LIN {X 0,Y 193.784,Z 1192.753,A -85,B 0,C 180,E1 2958.088,E2 2958.088} C_VEL
LIN {X 0,Y 196.55,Z 1189.097,A -85,B 0,C 180,E1 2951.921,E2 2951.921} C_VEL
LIN {X 0,Y 200.863,Z 1184.423,A -85,B 0,C 180,E1 2945.908,E2 2945.908} C_VEL
LIN {X 0,Y 207.135,Z 1178.405,A -85,B 0,C 180,E1 2939.865,E2 2939.865} C_VEL
LIN {X 0,Y 216.126,Z 1170.427,A -85,B 0,C 180,E1 2933.611,E2 2933.611} C_VEL
LIN {X 0,Y 228.412,Z 1159.714,A -85,B 0,C 180,E1 2927.271,E2 2927.271} C_VEL
LIN {X 0,Y 240.181,Z 1149.383,A -85,B 0,C 180,E1 2922.535,E2 2922.535} C_VEL
LIN {X 0,Y 252.062,Z 1138.725,A -85,B 0,C 180,E1 2918.605,E2 2918.605} C_VEL
LIN {X 0,Y 266.276,Z 1125.508,A -85,B 0,C 180,E1 2914.678,E2 2914.678} C_VEL
LIN {X 0,Y 283.027,Z 1108.844,A -85,B 0,C 180,E1 2910.815,E2 2910.815} C_VEL
LIN {X 0,Y 296.928,Z 1094.045,A -85,B 0,C 180,E1 2908.083,E2 2908.083} C_VEL
LIN {X 0,Y 310.128,Z 1079.059,A -85,B 0,C 180,E1 2905.802,E2 2905.802} C_VEL
LIN {X 0,Y 325.384,Z 1060.451,A -85,B 0,C 180,E1 2903.47,E2 2903.47} C_VEL
LIN {X 0,Y 340.885,Z 1039.444,A -85,B 0,C 180,E1 2901.363,E2 2901.363} C_VEL
LIN {X 0,Y 353.003,Z 1021.479,A -85,B 0,C 180,E1 2899.882,E2 2899.882} C_VEL
LIN {X 0,Y 363.602,Z 1004.327,A -85,B 0,C 180,E1 2898.674,E2 2898.674} C_VEL
LIN {X 0,Y 374.359,Z 985.261,A -85,B 0,C 180,E1 2897.538,E2 2897.538} C_VEL
LIN {X 0,Y 386.572,Z 961.109,A -85,B 0,C 180,E1 2896.341,E2 2896.341} C_VEL
LIN {X 0,Y 397.152,Z 936.648,A -85,B 0,C 180,E1 2895.366,E2 2895.366} C_VEL
LIN {X 0,Y 404.715,Z 916.743,A -85,B 0,C 180,E1 2894.708,E2 2894.708} C_VEL
LIN {X 0,Y 411.43,Z 896.473,A -85,B 0,C 180,E1 2894.146,E2 2894.146} C_VEL
LIN {X 0,Y 417.527,Z 874.884,A -85,B 0,C 180,E1 2893.651,E2 2893.651} C_VEL
LIN {X 0,Y 423.796,Z 847.505,A -85,B 0,C 180,E1 2893.158,E2 2893.158} C_VEL
LIN {X 0,Y 428.05,Z 821.26,A -85,B 0,C 180,E1 2892.768,E2 2892.768} C_VEL
LIN {X 0,Y 447.316,Z 647.119,A -85,B 0,C 180,E1 2890.414,E2 2890.414} C_VEL
LIN {X 0,Y 447.378,Z 646.28,A -85,B 0,C 180,E1 2890.372,E2 2890.372} C_VEL
LIN {X 0,Y 445.988,Z 643.083,A -85,B 0,C 180,E1 2888.25,E2 2888.25} C_VEL
LIN {X 0,Y 444.811,Z 639.498,A -85,B 0,C 180,E1 2884.758,E2 2884.758} C_VEL
LIN {X 0,Y 444.548,Z 640.357,A -85,B 0,C 180,E1 2883.764,E2 2883.764} C_VEL
LIN {X 0,Y 444.064,Z 644.495,A -85,B 0,C 180,E1 2882.115,E2 2882.115} C_VEL
LIN {X 0,Y 443.95,Z 648.203,A -85,B 0,C 180,E1 2880.587,E2 2880.587} C_VEL
LIN {X 0,Y 444,Z 648.603,A -85,B 0,C 180,E1 2880.301,E2 2880.301} C_VEL
LIN {X 0,Y 445.315,Z 651.864,A -85,B 0,C 180,E1 2877.297,E2 2877.297} C_VEL
LIN {X 0,Y 445.715,Z 653.234,A -85,B 0,C 180,E1 2876.601,E2 2876.601} C_VEL
LIN {X 0,Y 426.682,Z 822.591,A -85,B 0,C 180,E1 2874.347,E2 2874.347} C_VEL
LIN {X 0,Y 422.446,Z 848.515,A -85,B 0,C 180,E1 2873.967,E2 2873.967} C_VEL
LIN {X 0,Y 416.03,Z 876.307,A -85,B 0,C 180,E1 2873.503,E2 2873.503} C_VEL
LIN {X 0,Y 409.724,Z 898.303,A -85,B 0,C 180,E1 2873.036,E2 2873.036} C_VEL
LIN {X 0,Y 402.64,Z 919.334,A -85,B 0,C 180,E1 2872.488,E2 2872.488} C_VEL
LIN {X 0,Y 393.996,Z 941.562,A -85,B 0,C 180,E1 2871.786,E2 2871.786} C_VEL
LIN {X 0,Y 381.931,Z 968.144,A -85,B 0,C 180,E1 2870.742,E2 2870.742} C_VEL
LIN {X 0,Y 371.433,Z 988.383,A -85,B 0,C 180,E1 2869.766,E2 2869.766} C_VEL
LIN {X 0,Y 360.939,Z 1006.691,A -85,B 0,C 180,E1 2868.714,E2 2868.714} C_VEL
LIN {X 0,Y 349.835,Z 1024.338,A -85,B 0,C 180,E1 2867.527,E2 2867.527} C_VEL
LIN {X 0,Y 336.067,Z 1044.358,A -85,B 0,C 180,E1 2865.914,E2 2865.914} C_VEL
LIN {X 0,Y 319.422,Z 1066.078,A -85,B 0,C 180,E1 2863.734,E2 2863.734} C_VEL
LIN {X 0,Y 305.681,Z 1082.487,A -85,B 0,C 180,E1 2861.698,E2 2861.698} C_VEL
LIN {X 0,Y 292.491,Z 1097.171,A -85,B 0,C 180,E1 2859.501,E2 2859.501} C_VEL
LIN {X 0,Y 278.409,Z 1111.856,A -85,B 0,C 180,E1 2856.839,E2 2856.839} C_VEL
LIN {X 0,Y 260.253,Z 1129.443,A -85,B 0,C 180,E1 2852.794,E2 2852.794} C_VEL
LIN {X 0,Y 246.812,Z 1141.663,A -85,B 0,C 180,E1 2849.189,E2 2849.189} C_VEL
LIN {X 0,Y 234.676,Z 1152.282,A -85,B 0,C 180,E1 2845.318,E2 2845.318} C_VEL
LIN {X 0,Y 222.868,Z 1162.354,A -85,B 0,C 180,E1 2840.758,E2 2840.758} C_VEL
LIN {X 0,Y 210.031,Z 1173.278,A -85,B 0,C 180,E1 2834.413,E2 2834.413} C_VEL
LIN {X 0,Y 199.904,Z 1181.947,A -85,B 0,C 180,E1 2827.607,E2 2827.607} C_VEL
LIN {X 0,Y 193.365,Z 1187.998,A -85,B 0,C 180,E1 2821.485,E2 2821.485} C_VEL
LIN {X 0,Y 188.86,Z 1192.711,A -85,B 0,C 180,E1 2815.395,E2 2815.395} C_VEL
LIN {X 0,Y 185.836,Z 1196.591,A -85,B 0,C 180,E1 2808.835,E2 2808.835} C_VEL
LIN {X 0,Y 184.378,Z 1199.289,A -85,B 0,C 180,E1 2802.529,E2 2802.529} C_VEL
LIN {X 0,Y 183.967,Z 1200.898,A -85,B 0,C 180,E1 2796.869,E2 2796.869} C_VEL
LIN {X 0,Y 183.92,Z 1201.731,A -85,B 0,C 180,E1 2791.559,E2 2791.559} C_VEL
LIN {X 0,Y 183.915,Z 1201.914,A -85,B 0,C 180,E1 2786.261,E2 2786.261} C_VEL
LIN {X 0,Y 184.128,Z 1201.247,A -85,B 0,C 180,E1 2779.994,E2 2779.994} C_VEL
LIN {X 0,Y 185.319,Z 1199.444,A -85,B 0,C 180,E1 2773.062,E2 2773.062} C_VEL
LIN {X 0,Y 188.166,Z 1196.498,A -85,B 0,C 180,E1 2766.063,E2 2766.063} C_VEL
LIN {X 0,Y 192.831,Z 1192.57,A -85,B 0,C 180,E1 2759.46,E2 2759.46} C_VEL
LIN {X 0,Y 199.23,Z 1187.715,A -85,B 0,C 180,E1 2753.33,E2 2753.33} C_VEL
LIN {X 0,Y 208.339,Z 1181.197,A -85,B 0,C 180,E1 2747.041,E2 2747.041} C_VEL
LIN {X 0,Y 222.726,Z 1171.072,A -85,B 0,C 180,E1 2739.857,E2 2739.857} C_VEL
LIN {X 0,Y 236.169,Z 1161.389,A -85,B 0,C 180,E1 2734.782,E2 2734.782} C_VEL
LIN {X 0,Y 249.143,Z 1151.762,A -85,B 0,C 180,E1 2730.816,E2 2730.816} C_VEL
LIN {X 0,Y 263.881,Z 1140.338,A -85,B 0,C 180,E1 2727.073,E2 2727.073} C_VEL
LIN {X 0,Y 282.835,Z 1124.684,A -85,B 0,C 180,E1 2723.105,E2 2723.105} C_VEL
LIN {X 0,Y 299.39,Z 1109.822,A -85,B 0,C 180,E1 2720.208,E2 2720.208} C_VEL
LIN {X 0,Y 314.262,Z 1095.515,A -85,B 0,C 180,E1 2717.954,E2 2717.954} C_VEL
LIN {X 0,Y 329.586,Z 1079.656,A -85,B 0,C 180,E1 2715.913,E2 2715.913} C_VEL
LIN {X 0,Y 347.949,Z 1058.826,A -85,B 0,C 180,E1 2713.767,E2 2713.767} C_VEL
LIN {X 0,Y 362.448,Z 1040.568,A -85,B 0,C 180,E1 2712.264,E2 2712.264} C_VEL
LIN {X 0,Y 375.061,Z 1023.222,A -85,B 0,C 180,E1 2711.067,E2 2711.067} C_VEL
LIN {X 0,Y 387.331,Z 1004.748,A -85,B 0,C 180,E1 2710,E2 2710} C_VEL
LIN {X 0,Y 399.863,Z 983.893,A -85,B 0,C 180,E1 2708.994,E2 2708.994} C_VEL
LIN {X 0,Y 413.455,Z 958.023,A -85,B 0,C 180,E1 2707.988,E2 2707.988} C_VEL
LIN {X 0,Y 422.9,Z 937.408,A -85,B 0,C 180,E1 2707.335,E2 2707.335} C_VEL
LIN {X 0,Y 431.26,Z 916.643,A -85,B 0,C 180,E1 2706.791,E2 2706.791} C_VEL
LIN {X 0,Y 438.618,Z 895.545,A -85,B 0,C 180,E1 2706.334,E2 2706.334} C_VEL
LIN {X 0,Y 446.408,Z 868.875,A -85,B 0,C 180,E1 2705.874,E2 2705.874} C_VEL
LIN {X 0,Y 452.306,Z 842.166,A -85,B 0,C 180,E1 2705.505,E2 2705.505} C_VEL
LIN {X 0,Y 456.042,Z 819.713,A -85,B 0,C 180,E1 2705.211,E2 2705.211} C_VEL
LIN {X 0,Y 473.449,Z 676.945,A -85,B 0,C 180,E1 2703.423,E2 2703.423} C_VEL
LIN {X 0,Y 473.466,Z 676.653,A -85,B 0,C 180,E1 2702.713,E2 2702.713} C_VEL
LIN {X 0,Y 473.43,Z 677.084,A -85,B 0,C 180,E1 2702.407,E2 2702.407} C_VEL
LIN {X 0,Y 455.697,Z 821.974,A -85,B 0,C 180,E1 2700.598,E2 2700.598} C_VEL
LIN {X 0,Y 450.971,Z 849.012,A -85,B 0,C 180,E1 2700.243,E2 2700.243} C_VEL
LIN {X 0,Y 444.348,Z 875.944,A -85,B 0,C 180,E1 2699.835,E2 2699.835} C_VEL
LIN {X 0,Y 437.962,Z 897.143,A -85,B 0,C 180,E1 2699.43,E2 2699.43} C_VEL
LIN {X 0,Y 430.703,Z 917.681,A -85,B 0,C 180,E1 2698.954,E2 2698.954} C_VEL
LIN {X 0,Y 422.114,Z 938.76,A -85,B 0,C 180,E1 2698.367,E2 2698.367} C_VEL
LIN {X 0,Y 409.93,Z 964.599,A -85,B 0,C 180,E1 2697.484,E2 2697.484} C_VEL
LIN {X 0,Y 398.155,Z 986.144,A -85,B 0,C 180,E1 2696.577,E2 2696.577} C_VEL
LIN {X 0,Y 387.061,Z 1004.427,A -85,B 0,C 180,E1 2695.652,E2 2695.652} C_VEL
LIN {X 0,Y 375.114,Z 1022.302,A -85,B 0,C 180,E1 2694.599,E2 2694.599} C_VEL
LIN {X 0,Y 361.439,Z 1040.964,A -85,B 0,C 180,E1 2693.273,E2 2693.273} C_VEL
LIN {X 0,Y 343.377,Z 1063.103,A -85,B 0,C 180,E1 2691.329,E2 2691.329} C_VEL
LIN {X 0,Y 328.434,Z 1079.641,A -85,B 0,C 180,E1 2689.52,E2 2689.52} C_VEL
LIN {X 0,Y 314.281,Z 1094.13,A -85,B 0,C 180,E1 2687.606,E2 2687.606} C_VEL
LIN {X 0,Y 299.083,Z 1108.599,A -85,B 0,C 180,E1 2685.281,E2 2685.281} C_VEL
LIN {X 0,Y 280.33,Z 1125.143,A -85,B 0,C 180,E1 2681.922,E2 2681.922} C_VEL
LIN {X 0,Y 263.578,Z 1138.659,A -85,B 0,C 180,E1 2678.339,E2 2678.339} C_VEL
LIN {X 0,Y 249.729,Z 1149.238,A -85,B 0,C 180,E1 2674.803,E2 2674.803} C_VEL
LIN {X 0,Y 236.884,Z 1158.604,A -85,B 0,C 180,E1 2670.894,E2 2670.894} C_VEL
LIN {X 0,Y 223.454,Z 1168.069,A -85,B 0,C 180,E1 2665.872,E2 2665.872} C_VEL
LIN {X 0,Y 209.417,Z 1177.701,A -85,B 0,C 180,E1 2658.969,E2 2658.969} C_VEL
LIN {X 0,Y 200.157,Z 1184.082,A -85,B 0,C 180,E1 2652.748,E2 2652.748} C_VEL
LIN {X 0,Y 193.407,Z 1188.958,A -85,B 0,C 180,E1 2646.477,E2 2646.477} C_VEL
LIN {X 0,Y 188.589,Z 1192.766,A -85,B 0,C 180,E1 2639.891,E2 2639.891} C_VEL
LIN {X 0,Y 185.648,Z 1195.509,A -85,B 0,C 180,E1 2633.15,E2 2633.15} C_VEL
LIN {X 0,Y 184.261,Z 1197.282,A -85,B 0,C 180,E1 2626.065,E2 2626.065} C_VEL
LIN {X 0,Y 183.939,Z 1197.909,A -85,B 0,C 180,E1 2619.7,E2 2619.7} C_VEL
LIN {X 0,Y 183.918,Z 1197.682,A -85,B 0,C 180,E1 2614.052,E2 2614.052} C_VEL
LIN {X 0,Y 184.043,Z 1196.747,A -85,B 0,C 180,E1 2608.442,E2 2608.442} C_VEL
LIN {X 0,Y 184.659,Z 1194.997,A -85,B 0,C 180,E1 2602.532,E2 2602.532} C_VEL
LIN {X 0,Y 186.366,Z 1192.29,A -85,B 0,C 180,E1 2596.344,E2 2596.344} C_VEL
LIN {X 0,Y 189.631,Z 1188.474,A -85,B 0,C 180,E1 2589.956,E2 2589.956} C_VEL
LIN {X 0,Y 195.401,Z 1182.891,A -85,B 0,C 180,E1 2582.907,E2 2582.907} C_VEL
LIN {X 0,Y 204.952,Z 1174.56,A -85,B 0,C 180,E1 2575.193,E2 2575.193} C_VEL
LIN {X 0,Y 214.979,Z 1166.193,A -85,B 0,C 180,E1 2569.371,E2 2569.371} C_VEL
LIN {X 0,Y 225.673,Z 1157.324,A -85,B 0,C 180,E1 2564.492,E2 2564.492} C_VEL
LIN {X 0,Y 238.322,Z 1146.688,A -85,B 0,C 180,E1 2559.844,E2 2559.844} C_VEL
LIN {X 0,Y 254.991,Z 1132.046,A -85,B 0,C 180,E1 2554.925,E2 2554.925} C_VEL
LIN {X 0,Y 268.749,Z 1119.234,A -85,B 0,C 180,E1 2551.57,E2 2551.57} C_VEL
LIN {X 0,Y 281.856,Z 1106.336,A -85,B 0,C 180,E1 2548.808,E2 2548.808} C_VEL
LIN {X 0,Y 295.173,Z 1092.404,A -85,B 0,C 180,E1 2546.344,E2 2546.344} C_VEL
LIN {X 0,Y 311.307,Z 1074.339,A -85,B 0,C 180,E1 2543.739,E2 2543.739} C_VEL
LIN {X 0,Y 327.195,Z 1054.608,A -85,B 0,C 180,E1 2541.482,E2 2541.482} C_VEL
LIN {X 0,Y 340.141,Z 1037.088,A -85,B 0,C 180,E1 2539.834,E2 2539.834} C_VEL
LIN {X 0,Y 352.066,Z 1019.537,A -85,B 0,C 180,E1 2538.455,E2 2538.455} C_VEL
LIN {X 0,Y 364.175,Z 1000.011,A -85,B 0,C 180,E1 2537.162,E2 2537.162} C_VEL
LIN {X 0,Y 377.653,Z 975.504,A -85,B 0,C 180,E1 2535.826,E2 2535.826} C_VEL
LIN {X 0,Y 387.964,Z 954.171,A -85,B 0,C 180,E1 2534.879,E2 2534.879} C_VEL
LIN {X 0,Y 396.471,Z 934.374,A -85,B 0,C 180,E1 2534.143,E2 2534.143} C_VEL
LIN {X 0,Y 404.135,Z 914.142,A -85,B 0,C 180,E1 2533.509,E2 2533.509} C_VEL
LIN {X 0,Y 412.068,Z 889.833,A -85,B 0,C 180,E1 2532.879,E2 2532.879} C_VEL
LIN {X 0,Y 419.216,Z 862.435,A -85,B 0,C 180,E1 2532.33,E2 2532.33} C_VEL
LIN {X 0,Y 423.88,Z 839.666,A -85,B 0,C 180,E1 2531.97,E2 2531.97} C_VEL
LIN {X 0,Y 427.315,Z 817.269,A -85,B 0,C 180,E1 2531.649,E2 2531.649} C_VEL
LIN {X 0,Y 445.713,Z 652.932,A -85,B 0,C 180,E1 2529.458,E2 2529.458} C_VEL
LIN {X 0,Y 444.938,Z 650.967,A -85,B 0,C 180,E1 2528.139,E2 2528.139} C_VEL
LIN {X 0,Y 443.812,Z 647.425,A -85,B 0,C 180,E1 2524.652,E2 2524.652} C_VEL
LIN {X 0,Y 443.864,Z 647.551,A -85,B 0,C 180,E1 2521.162,E2 2521.162} C_VEL
LIN {X 0,Y 444,Z 648.603,A -85,B 0,C 180,E1 2520.301,E2 2520.301} C_VEL
LIN {X 0,Y 444.352,Z 650.816,A -85,B 0,C 180,E1 2518.94,E2 2518.94} C_VEL
LIN {X 0,Y 444.48,Z 653.384,A -85,B 0,C 180,E1 2518.202,E2 2518.202} C_VEL
LIN {X 0,Y 444.411,Z 656.348,A -85,B 0,C 180,E1 2517.767,E2 2517.767} C_VEL
LIN {X 0,Y 444.172,Z 659.579,A -85,B 0,C 180,E1 2517.547,E2 2517.547} C_VEL
LIN {X 0,Y 425.554,Z 822.606,A -85,B 0,C 180,E1 2515.415,E2 2515.415} C_VEL
LIN {X 0,Y 421.185,Z 848.96,A -85,B 0,C 180,E1 2515.039,E2 2515.039} C_VEL
LIN {X 0,Y 414.704,Z 876.574,A -85,B 0,C 180,E1 2514.592,E2 2514.592} C_VEL
LIN {X 0,Y 408.459,Z 898.118,A -85,B 0,C 180,E1 2514.152,E2 2514.152} C_VEL
LIN {X 0,Y 401.429,Z 918.8,A -85,B 0,C 180,E1 2513.634,E2 2513.634} C_VEL
LIN {X 0,Y 392.432,Z 941.7,A -85,B 0,C 180,E1 2512.937,E2 2512.937} C_VEL
LIN {X 0,Y 380.221,Z 968.234,A -85,B 0,C 180,E1 2511.93,E2 2511.93} C_VEL
LIN {X 0,Y 369.526,Z 988.564,A -85,B 0,C 180,E1 2510.981,E2 2510.981} C_VEL
LIN {X 0,Y 358.884,Z 1006.85,A -85,B 0,C 180,E1 2509.961,E2 2509.961} C_VEL
LIN {X 0,Y 347.571,Z 1024.544,A -85,B 0,C 180,E1 2508.808,E2 2508.808} C_VEL
LIN {X 0,Y 332.902,Z 1045.5,A -85,B 0,C 180,E1 2507.158,E2 2507.158} C_VEL
LIN {X 0,Y 316.333,Z 1066.583,A -85,B 0,C 180,E1 2505.075,E2 2505.075} C_VEL
LIN {X 0,Y 302.936,Z 1082.257,A -85,B 0,C 180,E1 2503.174,E2 2503.174} C_VEL
LIN {X 0,Y 289.651,Z 1096.737,A -85,B 0,C 180,E1 2501.06,E2 2501.06} C_VEL
LIN {X 0,Y 275.986,Z 1110.665,A -85,B 0,C 180,E1 2498.607,E2 2498.607} C_VEL
LIN {X 0,Y 259.115,Z 1126.81,A -85,B 0,C 180,E1 2495.071,E2 2495.071} C_VEL
LIN {X 0,Y 242.557,Z 1141.372,A -85,B 0,C 180,E1 2490.894,E2 2490.894} C_VEL
LIN {X 0,Y 229.971,Z 1151.986,A -85,B 0,C 180,E1 2487.05,E2 2487.05} C_VEL
LIN {X 0,Y 217.832,Z 1161.904,A -85,B 0,C 180,E1 2482.571,E2 2482.571} C_VEL
LIN {X 0,Y 204.987,Z 1172.328,A -85,B 0,C 180,E1 2476.546,E2 2476.546} C_VEL
LIN {X 0,Y 193.711,Z 1181.428,A -85,B 0,C 180,E1 2469.413,E2 2469.413} C_VEL
LIN {X 0,Y 186.602,Z 1187.549,A -85,B 0,C 180,E1 2463.132,E2 2463.132} C_VEL
LIN {X 0,Y 181.412,Z 1192.542,A -85,B 0,C 180,E1 2456.517,E2 2456.517} C_VEL
LIN {X 0,Y 178.201,Z 1196.278,A -85,B 0,C 180,E1 2450.016,E2 2450.016} C_VEL
LIN {X 0,Y 176.553,Z 1198.926,A -85,B 0,C 180,E1 2443.761,E2 2443.761} C_VEL
LIN {X 0,Y 176.006,Z 1200.647,A -85,B 0,C 180,E1 2437.837,E2 2437.837} C_VEL
LIN {X 0,Y 175.916,Z 1201.59,A -85,B 0,C 180,E1 2432.281,E2 2432.281} C_VEL
LIN {X 0,Y 175.915,Z 1201.858,A -85,B 0,C 180,E1 2426.417,E2 2426.417} C_VEL
LIN {X 0,Y 176.136,Z 1201.253,A -85,B 0,C 180,E1 2419.866,E2 2419.866} C_VEL
LIN {X 0,Y 177.562,Z 1199.335,A -85,B 0,C 180,E1 2412.116,E2 2412.116} C_VEL
LIN {X 0,Y 180.772,Z 1196.365,A -85,B 0,C 180,E1 2404.794,E2 2404.794} C_VEL
LIN {X 0,Y 185.712,Z 1192.557,A -85,B 0,C 180,E1 2398.156,E2 2398.156} C_VEL
LIN {X 0,Y 192.592,Z 1187.722,A -85,B 0,C 180,E1 2391.845,E2 2391.845} C_VEL
LIN {X 0,Y 201.817,Z 1181.526,A -85,B 0,C 180,E1 2385.69,E2 2385.69} C_VEL
LIN {X 0,Y 215.739,Z 1172.347,A -85,B 0,C 180,E1 2378.867,E2 2378.867} C_VEL
LIN {X 0,Y 230.84,Z 1161.935,A -85,B 0,C 180,E1 2373.285,E2 2373.285} C_VEL
LIN {X 0,Y 244.956,Z 1151.875,A -85,B 0,C 180,E1 2369.132,E2 2369.132} C_VEL
LIN {X 0,Y 259.673,Z 1140.865,A -85,B 0,C 180,E1 2365.548,E2 2365.548} C_VEL
LIN {X 0,Y 277.939,Z 1126.377,A -85,B 0,C 180,E1 2361.855,E2 2361.855} C_VEL
LIN {X 0,Y 296.631,Z 1110.043,A -85,B 0,C 180,E1 2358.707,E2 2358.707} C_VEL
LIN {X 0,Y 311.816,Z 1095.77,A -85,B 0,C 180,E1 2356.511,E2 2356.511} C_VEL
LIN {X 0,Y 326.549,Z 1080.856,A -85,B 0,C 180,E1 2354.634,E2 2354.634} C_VEL
LIN {X 0,Y 343.701,Z 1062.031,A -85,B 0,C 180,E1 2352.707,E2 2352.707} C_VEL
LIN {X 0,Y 360.601,Z 1041.239,A -85,B 0,C 180,E1 2351.021,E2 2351.021} C_VEL
LIN {X 0,Y 373.464,Z 1023.85,A -85,B 0,C 180,E1 2349.859,E2 2349.859} C_VEL
LIN {X 0,Y 386.012,Z 1005.253,A -85,B 0,C 180,E1 2348.82,E2 2348.82} C_VEL
LIN {X 0,Y 398.151,Z 985.373,A -85,B 0,C 180,E1 2347.892,E2 2347.892} C_VEL
LIN {X 0,Y 411.946,Z 959.743,A -85,B 0,C 180,E1 2346.921,E2 2346.921} C_VEL
LIN {X 0,Y 422.054,Z 938.014,A -85,B 0,C 180,E1 2346.256,E2 2346.256} C_VEL
LIN {X 0,Y 430.556,Z 917.171,A -85,B 0,C 180,E1 2345.731,E2 2345.731} C_VEL
LIN {X 0,Y 437.815,Z 896.656,A -85,B 0,C 180,E1 2345.303,E2 2345.303} C_VEL
LIN {X 0,Y 444.69,Z 873.748,A -85,B 0,C 180,E1 2344.916,E2 2344.916} C_VEL
LIN {X 0,Y 451.59,Z 844.325,A -85,B 0,C 180,E1 2344.515,E2 2344.515} C_VEL
LIN {X 0,Y 455.609,Z 820.905,A -85,B 0,C 180,E1 2344.216,E2 2344.216} C_VEL
LIN {X 0,Y 468.719,Z 715.222,A -85,B 0,C 180,E1 2342.917,E2 2342.917} C_VEL
LIN {X 0,Y 455.367,Z 822.493,A -85,B 0,C 180,E1 2341.602,E2 2341.602} C_VEL
LIN {X 0,Y 450.457,Z 850.026,A -85,B 0,C 180,E1 2341.25,E2 2341.25} C_VEL
LIN {X 0,Y 443.865,Z 876.418,A -85,B 0,C 180,E1 2340.865,E2 2340.865} C_VEL
LIN {X 0,Y 437.456,Z 897.463,A -85,B 0,C 180,E1 2340.479,E2 2340.479} C_VEL
LIN {X 0,Y 429.941,Z 918.467,A -85,B 0,C 180,E1 2340.01,E2 2340.01} C_VEL
LIN {X 0,Y 420.964,Z 940.178,A -85,B 0,C 180,E1 2339.426,E2 2339.426} C_VEL
LIN {X 0,Y 408.077,Z 966.828,A -85,B 0,C 180,E1 2338.537,E2 2338.537} C_VEL
LIN {X 0,Y 396.763,Z 987.176,A -85,B 0,C 180,E1 2337.705,E2 2337.705} C_VEL
LIN {X 0,Y 385.543,Z 1005.357,A -85,B 0,C 180,E1 2336.815,E2 2336.815} C_VEL
LIN {X 0,Y 372.971,Z 1023.834,A -85,B 0,C 180,E1 2335.756,E2 2335.756} C_VEL
LIN {X 0,Y 356.752,Z 1045.434,A -85,B 0,C 180,E1 2334.239,E2 2334.239} C_VEL
LIN {X 0,Y 339.871,Z 1065.317,A -85,B 0,C 180,E1 2332.486,E2 2332.486} C_VEL
LIN {X 0,Y 325.458,Z 1080.893,A -85,B 0,C 180,E1 2330.807,E2 2330.807} C_VEL
LIN {X 0,Y 311.659,Z 1094.696,A -85,B 0,C 180,E1 2329.023,E2 2329.023} C_VEL
LIN {X 0,Y 295.88,Z 1109.358,A -85,B 0,C 180,E1 2326.713,E2 2326.713} C_VEL
LIN {X 0,Y 275.685,Z 1126.571,A -85,B 0,C 180,E1 2323.232,E2 2323.232} C_VEL
LIN {X 0,Y 259.719,Z 1139.063,A -85,B 0,C 180,E1 2319.942,E2 2319.942} C_VEL
LIN {X 0,Y 245.419,Z 1149.607,A -85,B 0,C 180,E1 2316.443,E2 2316.443} C_VEL
LIN {X 0,Y 231.427,Z 1159.409,A -85,B 0,C 180,E1 2312.335,E2 2312.335} C_VEL
LIN {X 0,Y 215.672,Z 1170.022,A -85,B 0,C 180,E1 2306.516,E2 2306.516} C_VEL
LIN {X 0,Y 202.351,Z 1178.566,A -85,B 0,C 180,E1 2299.985,E2 2299.985} C_VEL
LIN {X 0,Y 193.156,Z 1184.533,A -85,B 0,C 180,E1 2293.918,E2 2293.918} C_VEL
LIN {X 0,Y 185.98,Z 1189.365,A -85,B 0,C 180,E1 2287.408,E2 2287.408} C_VEL
LIN {X 0,Y 180.489,Z 1193.42,A -85,B 0,C 180,E1 2279.905,E2 2279.905} C_VEL
LIN {X 0,Y 177.091,Z 1196.472,A -85,B 0,C 180,E1 2271.182,E2 2271.182} C_VEL
LIN {X 0,Y 176.073,Z 1197.751,A -85,B 0,C 180,E1 2263.797,E2 2263.797} C_VEL
LIN {X 0,Y 175.934,Z 1198.011,A -85,B 0,C 180,E1 2257.51,E2 2257.51} C_VEL
LIN {X 0,Y 175.946,Z 1197.472,A -85,B 0,C 180,E1 2251.301,E2 2251.301} C_VEL
LIN {X 0,Y 176.364,Z 1195.919,A -85,B 0,C 180,E1 2244.468,E2 2244.468} C_VEL
LIN {X 0,Y 178.067,Z 1193.078,A -85,B 0,C 180,E1 2237.019,E2 2237.019} C_VEL
LIN {X 0,Y 181.448,Z 1189.265,A -85,B 0,C 180,E1 2230.021,E2 2230.021} C_VEL
LIN {X 0,Y 186.444,Z 1184.59,A -85,B 0,C 180,E1 2223.568,E2 2223.568} C_VEL
LIN {X 0,Y 193.236,Z 1178.865,A -85,B 0,C 180,E1 2217.442,E2 2217.442} C_VEL
LIN {X 0,Y 202.214,Z 1171.705,A -85,B 0,C 180,E1 2211.461,E2 2211.461} C_VEL
LIN {X 0,Y 215.622,Z 1161.215,A -85,B 0,C 180,E1 2204.805,E2 2204.805} C_VEL
LIN {X 0,Y 228.848,Z 1150.539,A -85,B 0,C 180,E1 2199.737,E2 2199.737} C_VEL
LIN {X 0,Y 241.557,Z 1139.991,A -85,B 0,C 180,E1 2195.775,E2 2195.775} C_VEL
LIN {X 0,Y 255.262,Z 1128.1,A -85,B 0,C 180,E1 2192.19,E2 2192.19} C_VEL
LIN {X 0,Y 271.975,Z 1112.783,A -85,B 0,C 180,E1 2188.519,E2 2188.519} C_VEL
LIN {X 0,Y 288.864,Z 1095.811,A -85,B 0,C 180,E1 2185.386,E2 2185.386} C_VEL
LIN {X 0,Y 302.905,Z 1080.658,A -85,B 0,C 180,E1 2183.13,E2 2183.13} C_VEL
LIN {X 0,Y 316.385,Z 1065.003,A -85,B 0,C 180,E1 2181.203,E2 2181.203} C_VEL
LIN {X 0,Y 332.388,Z 1044.844,A -85,B 0,C 180,E1 2179.166,E2 2179.166} C_VEL
LIN {X 0,Y 347.442,Z 1023.48,A -85,B 0,C 180,E1 2177.445,E2 2177.445} C_VEL
LIN {X 0,Y 358.802,Z 1005.78,A -85,B 0,C 180,E1 2176.255,E2 2176.255} C_VEL
LIN {X 0,Y 369.863,Z 986.837,A -85,B 0,C 180,E1 2175.179,E2 2175.179} C_VEL
LIN {X 0,Y 381.047,Z 965.549,A -85,B 0,C 180,E1 2174.168,E2 2174.168} C_VEL
LIN {X 0,Y 393.246,Z 938.754,A -85,B 0,C 180,E1 2173.137,E2 2173.137} C_VEL
LIN {X 0,Y 401.445,Z 917.847,A -85,B 0,C 180,E1 2172.483,E2 2172.483} C_VEL
LIN {X 0,Y 408.543,Z 896.99,A -85,B 0,C 180,E1 2171.941,E2 2171.941} C_VEL
LIN {X 0,Y 414.836,Z 875.242,A -85,B 0,C 180,E1 2171.474,E2 2171.474} C_VEL
LIN {X 0,Y 421.213,Z 848.109,A -85,B 0,C 180,E1 2171.016,E2 2171.016} C_VEL
LIN {X 0,Y 425.643,Z 821.479,A -85,B 0,C 180,E1 2170.64,E2 2170.64} C_VEL
LIN {X 0,Y 444.16,Z 659.46,A -85,B 0,C 180,E1 2168.521,E2 2168.521} C_VEL
LIN {X 0,Y 442.813,Z 655.352,A -85,B 0,C 180,E1 2164.533,E2 2164.533} C_VEL
LIN {X 0,Y 442.874,Z 655.59,A -85,B 0,C 180,E1 2161.164,E2 2161.164} C_VEL
LIN {X 0,Y 444.172,Z 659.579,A -85,B 0,C 180,E1 2157.547,E2 2157.547} C_VEL
LIN {X 0,Y 443.559,Z 665.003,A -85,B 0,C 180,E1 2157.47,E2 2157.47} C_VEL
LIN {X 0,Y 442.514,Z 672.639,A -85,B 0,C 180,E1 2157.607,E2 2157.607} C_VEL
LIN {X 0,Y 440.292,Z 687.836,A -85,B 0,C 180,E1 2158.104,E2 2158.104} C_VEL
LIN {X 0,Y 439.447,Z 694.511,A -85,B 0,C 180,E1 2158.137,E2 2158.137} C_VEL
LIN {X 0,Y 424.554,Z 822.776,A -85,B 0,C 180,E1 2156.487,E2 2156.487} C_VEL
LIN {X 0,Y 419.951,Z 850.057,A -85,B 0,C 180,E1 2156.107,E2 2156.107} C_VEL
LIN {X 0,Y 413.468,Z 877.061,A -85,B 0,C 180,E1 2155.684,E2 2155.684} C_VEL
LIN {X 0,Y 407.096,Z 898.728,A -85,B 0,C 180,E1 2155.257,E2 2155.257} C_VEL
LIN {X 0,Y 399.641,Z 920.282,A -85,B 0,C 180,E1 2154.732,E2 2154.732} C_VEL
LIN {X 0,Y 389.598,Z 945.289,A -85,B 0,C 180,E1 2153.986,E2 2153.986} C_VEL
LIN {X 0,Y 378.01,Z 969.62,A -85,B 0,C 180,E1 2153.074,E2 2153.074} C_VEL
LIN {X 0,Y 367.484,Z 989.281,A -85,B 0,C 180,E1 2152.181,E2 2152.181} C_VEL
LIN {X 0,Y 356.804,Z 1007.327,A -85,B 0,C 180,E1 2151.204,E2 2151.204} C_VEL
LIN {X 0,Y 344.676,Z 1025.948,A -85,B 0,C 180,E1 2150.02,E2 2150.02} C_VEL
LIN {X 0,Y 328.792,Z 1048.011,A -85,B 0,C 180,E1 2148.302,E2 2148.302} C_VEL
LIN {X 0,Y 313.427,Z 1067.082,A -85,B 0,C 180,E1 2146.444,E2 2146.444} C_VEL
LIN {X 0,Y 299.752,Z 1082.735,A -85,B 0,C 180,E1 2144.584,E2 2144.584} C_VEL
LIN {X 0,Y 286.177,Z 1097.18,A -85,B 0,C 180,E1 2142.513,E2 2142.513} C_VEL
LIN {X 0,Y 269.801,Z 1113.414,A -85,B 0,C 180,E1 2139.656,E2 2139.656} C_VEL
LIN {X 0,Y 251.846,Z 1129.712,A -85,B 0,C 180,E1 2135.945,E2 2135.945} C_VEL
LIN {X 0,Y 237.696,Z 1141.758,A -85,B 0,C 180,E1 2132.437,E2 2132.437} C_VEL
LIN {X 0,Y 224.821,Z 1152.215,A -85,B 0,C 180,E1 2128.641,E2 2128.641} C_VEL
LIN {X 0,Y 211.604,Z 1162.57,A -85,B 0,C 180,E1 2123.904,E2 2123.904} C_VEL
LIN {X 0,Y 197.165,Z 1173.665,A -85,B 0,C 180,E1 2117.19,E2 2117.19} C_VEL
LIN {X 0,Y 186.405,Z 1181.905,A -85,B 0,C 180,E1 2110.386,E2 2110.386} C_VEL
LIN {X 0,Y 179.044,Z 1187.881,A -85,B 0,C 180,E1 2103.95,E2 2103.95} C_VEL
LIN {X 0,Y 173.6,Z 1192.796,A -85,B 0,C 180,E1 2097.067,E2 2097.067} C_VEL
LIN {X 0,Y 170,Z 1196.783,A -85,B 0,C 180,E1 2089.589,E2 2089.589} C_VEL
LIN {X 0,Y 168.225,Z 1199.855,A -85,B 0,C 180,E1 2081.267,E2 2081.267} C_VEL
LIN {X 0,Y 167.921,Z 1201.293,A -85,B 0,C 180,E1 2074.441,E2 2074.441} C_VEL
LIN {X 0,Y 167.916,Z 1201.762,A -85,B 0,C 180,E1 2068.295,E2 2068.295} C_VEL
LIN {X 0,Y 168.018,Z 1201.466,A -85,B 0,C 180,E1 2061.79,E2 2061.79} C_VEL
LIN {X 0,Y 169.053,Z 1200.071,A -85,B 0,C 180,E1 2053.861,E2 2053.861} C_VEL
LIN {X 0,Y 172.796,Z 1196.76,A -85,B 0,C 180,E1 2044.516,E2 2044.516} C_VEL
LIN {X 0,Y 178.395,Z 1192.753,A -85,B 0,C 180,E1 2037.068,E2 2037.068} C_VEL
LIN {X 0,Y 186.091,Z 1187.729,A -85,B 0,C 180,E1 2030.255,E2 2030.255} C_VEL
LIN {X 0,Y 195.955,Z 1181.52,A -85,B 0,C 180,E1 2023.945,E2 2023.945} C_VEL
LIN {X 0,Y 210.58,Z 1172.411,A -85,B 0,C 180,E1 2017.087,E2 2017.087} C_VEL
LIN {X 0,Y 227.014,Z 1161.571,A -85,B 0,C 180,E1 2011.301,E2 2011.301} C_VEL
LIN {X 0,Y 240.992,Z 1151.991,A -85,B 0,C 180,E1 2007.393,E2 2007.393} C_VEL
LIN {X 0,Y 255.937,Z 1141.185,A -85,B 0,C 180,E1 2003.914,E2 2003.914} C_VEL
LIN {X 0,Y 274.135,Z 1127.176,A -85,B 0,C 180,E1 2000.387,E2 2000.387} C_VEL
LIN {X 0,Y 293.232,Z 1111.029,A -85,B 0,C 180,E1 1997.304,E2 1997.304} C_VEL
LIN {X 0,Y 308.701,Z 1096.859,A -85,B 0,C 180,E1 1995.16,E2 1995.16} C_VEL
LIN {X 0,Y 323.679,Z 1082.056,A -85,B 0,C 180,E1 1993.332,E2 1993.332} C_VEL
LIN {X 0,Y 338.515,Z 1066.18,A -85,B 0,C 180,E1 1991.723,E2 1991.723} C_VEL
LIN {X 0,Y 355.444,Z 1046.408,A -85,B 0,C 180,E1 1990.086,E2 1990.086} C_VEL
LIN {X 0,Y 371.228,Z 1025.623,A -85,B 0,C 180,E1 1988.707,E2 1988.707} C_VEL
LIN {X 0,Y 383.913,Z 1007.216,A -85,B 0,C 180,E1 1987.705,E2 1987.705} C_VEL
LIN {X 0,Y 395.286,Z 989.039,A -85,B 0,C 180,E1 1986.872,E2 1986.872} C_VEL
LIN {X 0,Y 406.263,Z 969.594,A -85,B 0,C 180,E1 1986.124,E2 1986.124} C_VEL
LIN {X 0,Y 418.324,Z 945.545,A -85,B 0,C 180,E1 1985.363,E2 1985.363} C_VEL
LIN {X 0,Y 428.903,Z 920.557,A -85,B 0,C 180,E1 1984.731,E2 1984.731} C_VEL
LIN {X 0,Y 436.526,Z 899.643,A -85,B 0,C 180,E1 1984.303,E2 1984.303} C_VEL
LIN {X 0,Y 443.086,Z 878.547,A -85,B 0,C 180,E1 1983.951,E2 1983.951} C_VEL
LIN {X 0,Y 448.817,Z 856.333,A -85,B 0,C 180,E1 1983.647,E2 1983.647} C_VEL
LIN {X 0,Y 454.43,Z 828.173,A -85,B 0,C 180,E1 1983.294,E2 1983.294} C_VEL
LIN {X 0,Y 458.612,Z 797.4,A -85,B 0,C 180,E1 1982.916,E2 1982.916} C_VEL
LIN {X 0,Y 453.488,Z 833.501,A -85,B 0,C 180,E1 1982.478,E2 1982.478} C_VEL
LIN {X 0,Y 448.414,Z 857.94,A -85,B 0,C 180,E1 1982.171,E2 1982.171} C_VEL
LIN {X 0,Y 442.765,Z 879.553,A -85,B 0,C 180,E1 1981.854,E2 1981.854} C_VEL
LIN {X 0,Y 436.084,Z 900.81,A -85,B 0,C 180,E1 1981.469,E2 1981.469} C_VEL
LIN {X 0,Y 426.494,Z 926.58,A -85,B 0,C 180,E1 1980.894,E2 1980.894} C_VEL
LIN {X 0,Y 415.446,Z 951.159,A -85,B 0,C 180,E1 1980.205,E2 1980.205} C_VEL
LIN {X 0,Y 405.458,Z 970.728,A -85,B 0,C 180,E1 1979.538,E2 1979.538} C_VEL
LIN {X 0,Y 394.537,Z 989.868,A -85,B 0,C 180,E1 1978.769,E2 1978.769} C_VEL
LIN {X 0,Y 382.222,Z 1009.304,A -85,B 0,C 180,E1 1977.83,E2 1977.83} C_VEL
LIN {X 0,Y 365.646,Z 1032.587,A -85,B 0,C 180,E1 1976.462,E2 1976.462} C_VEL
LIN {X 0,Y 351.209,Z 1050.685,A -85,B 0,C 180,E1 1975.15,E2 1975.15} C_VEL
LIN {X 0,Y 336.753,Z 1067.262,A -85,B 0,C 180,E1 1973.693,E2 1973.693} C_VEL
LIN {X 0,Y 322.515,Z 1082.281,A -85,B 0,C 180,E1 1972.101,E2 1972.101} C_VEL
LIN {X 0,Y 305.622,Z 1098.709,A -85,B 0,C 180,E1 1969.978,E2 1969.978} C_VEL
LIN {X 0,Y 285.664,Z 1116.264,A -85,B 0,C 180,E1 1967.055,E2 1967.055} C_VEL
LIN {X 0,Y 269.961,Z 1128.951,A -85,B 0,C 180,E1 1964.358,E2 1964.358} C_VEL
LIN {X 0,Y 254.478,Z 1140.635,A -85,B 0,C 180,E1 1961.245,E2 1961.245} C_VEL
LIN {X 0,Y 237.959,Z 1152.338,A -85,B 0,C 180,E1 1957.258,E2 1957.258} C_VEL
LIN {X 0,Y 219.348,Z 1164.579,A -85,B 0,C 180,E1 1951.612,E2 1951.612} C_VEL
LIN {X 0,Y 206.077,Z 1172.877,A -85,B 0,C 180,E1 1946.418,E2 1946.418} C_VEL
LIN {X 0,Y 194.852,Z 1179.738,A -85,B 0,C 180,E1 1940.79,E2 1940.79} C_VEL
LIN {X 0,Y 184.581,Z 1186.042,A -85,B 0,C 180,E1 1933.896,E2 1933.896} C_VEL
LIN {X 0,Y 175.485,Z 1191.838,A -85,B 0,C 180,E1 1924.733,E2 1924.733} C_VEL
LIN {X 0,Y 171.028,Z 1195.019,A -85,B 0,C 180,E1 1917.128,E2 1917.128} C_VEL
LIN {X 0,Y 168.838,Z 1196.931,A -85,B 0,C 180,E1 1910.088,E2 1910.088} C_VEL
LIN {X 0,Y 168.07,Z 1197.872,A -85,B 0,C 180,E1 1903.765,E2 1903.765} C_VEL
LIN {X 0,Y 167.934,Z 1198.087,A -85,B 0,C 180,E1 1897.525,E2 1897.525} C_VEL
LIN {X 0,Y 167.945,Z 1197.591,A -85,B 0,C 180,E1 1891.363,E2 1891.363} C_VEL
LIN {X 0,Y 168.393,Z 1196.059,A -85,B 0,C 180,E1 1884.205,E2 1884.205} C_VEL
LIN {X 0,Y 170.235,Z 1193.24,A -85,B 0,C 180,E1 1876.411,E2 1876.411} C_VEL
LIN {X 0,Y 173.871,Z 1189.449,A -85,B 0,C 180,E1 1869.111,E2 1869.111} C_VEL
LIN {X 0,Y 179.214,Z 1184.797,A -85,B 0,C 180,E1 1862.413,E2 1862.413} C_VEL
LIN {X 0,Y 186.432,Z 1179.094,A -85,B 0,C 180,E1 1856.097,E2 1856.097} C_VEL
LIN {X 0,Y 195.954,Z 1171.916,A -85,B 0,C 180,E1 1849.943,E2 1849.943} C_VEL
LIN {X 0,Y 209.95,Z 1161.515,A -85,B 0,C 180,E1 1843.225,E2 1843.225} C_VEL
LIN {X 0,Y 224.349,Z 1150.36,A -85,B 0,C 180,E1 1837.92,E2 1837.92} C_VEL
LIN {X 0,Y 237.566,Z 1139.779,A -85,B 0,C 180,E1 1833.988,E2 1833.988} C_VEL
LIN {X 0,Y 251.71,Z 1127.885,A -85,B 0,C 180,E1 1830.457,E2 1830.457} C_VEL
LIN {X 0,Y 268.962,Z 1112.487,A -85,B 0,C 180,E1 1826.846,E2 1826.846} C_VEL
LIN {X 0,Y 286.29,Z 1095.447,A -85,B 0,C 180,E1 1823.787,E2 1823.787} C_VEL
LIN {X 0,Y 300.161,Z 1080.783,A -85,B 0,C 180,E1 1821.659,E2 1821.659} C_VEL
LIN {X 0,Y 314.4,Z 1064.547,A -85,B 0,C 180,E1 1819.718,E2 1819.718} C_VEL
LIN {X 0,Y 330.697,Z 1044.292,A -85,B 0,C 180,E1 1817.745,E2 1817.745} C_VEL
LIN {X 0,Y 345.57,Z 1023.478,A -85,B 0,C 180,E1 1816.127,E2 1816.127} C_VEL
LIN {X 0,Y 357.094,Z 1005.779,A -85,B 0,C 180,E1 1814.979,E2 1814.979} C_VEL
LIN {X 0,Y 368.304,Z 986.826,A -85,B 0,C 180,E1 1813.939,E2 1813.939} C_VEL
LIN {X 0,Y 379.633,Z 965.524,A -85,B 0,C 180,E1 1812.964,E2 1812.964} C_VEL
LIN {X 0,Y 391.52,Z 939.807,A -85,B 0,C 180,E1 1812.007,E2 1812.007} C_VEL
LIN {X 0,Y 400.14,Z 918.123,A -85,B 0,C 180,E1 1811.351,E2 1811.351} C_VEL
LIN {X 0,Y 407.213,Z 897.611,A -85,B 0,C 180,E1 1810.835,E2 1810.835} C_VEL
LIN {X 0,Y 413.44,Z 876.434,A -85,B 0,C 180,E1 1810.394,E2 1810.394} C_VEL
LIN {X 0,Y 419.458,Z 851.573,A -85,B 0,C 180,E1 1809.982,E2 1809.982} C_VEL
LIN {X 0,Y 424.457,Z 823.095,A -85,B 0,C 180,E1 1809.587,E2 1809.587} C_VEL
LIN {X 0,Y 433.375,Z 747.251,A -85,B 0,C 180,E1 1808.606,E2 1808.606} C_VEL
LIN {X 0,Y 442.66,Z 666.416,A -85,B 0,C 180,E1 1807.564,E2 1807.564} C_VEL
LIN {X 0,Y 441.838,Z 663.294,A -85,B 0,C 180,E1 1804.543,E2 1804.543} C_VEL
LIN {X 0,Y 441.873,Z 663.465,A -85,B 0,C 180,E1 1801.297,E2 1801.297} C_VEL
LIN {X 0,Y 442.663,Z 666.638,A -85,B 0,C 180,E1 1798.49,E2 1798.49} C_VEL
LIN {X 0,Y 439.447,Z 694.511,A -85,B 0,C 180,E1 1798.137,E2 1798.137} C_VEL
LIN {X 0,Y 438.476,Z 702.211,A -85,B 0,C 180,E1 1798.168,E2 1798.168} C_VEL
LIN {X 0,Y 435.592,Z 722.83,A -85,B 0,C 180,E1 1798.727,E2 1798.727} C_VEL
LIN {X 0,Y 434.767,Z 729.438,A -85,B 0,C 180,E1 1798.744,E2 1798.744} C_VEL
LIN {X 0,Y 423.638,Z 823.358,A -85,B 0,C 180,E1 1797.558,E2 1797.558} C_VEL
LIN {X 0,Y 418.801,Z 851.226,A -85,B 0,C 180,E1 1797.18,E2 1797.18} C_VEL
LIN {X 0,Y 412.444,Z 877.324,A -85,B 0,C 180,E1 1796.785,E2 1796.785} C_VEL
LIN {X 0,Y 406.134,Z 898.567,A -85,B 0,C 180,E1 1796.385,E2 1796.385} C_VEL
LIN {X 0,Y 398.575,Z 920.213,A -85,B 0,C 180,E1 1795.88,E2 1795.88} C_VEL
LIN {X 0,Y 388.34,Z 945.413,A -85,B 0,C 180,E1 1795.159,E2 1795.159} C_VEL
LIN {X 0,Y 376.46,Z 970.025,A -85,B 0,C 180,E1 1794.271,E2 1794.271} C_VEL
LIN {X 0,Y 366.345,Z 988.705,A -85,B 0,C 180,E1 1793.455,E2 1793.455} C_VEL
LIN {X 0,Y 355.488,Z 1006.853,A -85,B 0,C 180,E1 1792.515,E2 1792.515} C_VEL
LIN {X 0,Y 343.329,Z 1025.304,A -85,B 0,C 180,E1 1791.391,E2 1791.391} C_VEL
LIN {X 0,Y 327.2,Z 1047.46,A -85,B 0,C 180,E1 1789.735,E2 1789.735} C_VEL
LIN {X 0,Y 311.364,Z 1066.807,A -85,B 0,C 180,E1 1787.916,E2 1787.916} C_VEL
LIN {X 0,Y 297.274,Z 1082.648,A -85,B 0,C 180,E1 1786.094,E2 1786.094} C_VEL
LIN {X 0,Y 282.835,Z 1097.679,A -85,B 0,C 180,E1 1783.993,E2 1783.993} C_VEL
LIN {X 0,Y 265.343,Z 1114.583,A -85,B 0,C 180,E1 1781.056,E2 1781.056} C_VEL
LIN {X 0,Y 247.742,Z 1130.012,A -85,B 0,C 180,E1 1777.555,E2 1777.555} C_VEL
LIN {X 0,Y 233.36,Z 1141.87,A -85,B 0,C 180,E1 1774.132,E2 1774.132} C_VEL
LIN {X 0,Y 219.715,Z 1152.549,A -85,B 0,C 180,E1 1770.261,E2 1770.261} C_VEL
LIN {X 0,Y 205.411,Z 1163.3,A -85,B 0,C 180,E1 1765.282,E2 1765.282} C_VEL
LIN {X 0,Y 190.142,Z 1174.396,A -85,B 0,C 180,E1 1758.308,E2 1758.308} C_VEL
LIN {X 0,Y 179.578,Z 1182.071,A -85,B 0,C 180,E1 1751.745,E2 1751.745} C_VEL
LIN {X 0,Y 171.854,Z 1187.952,A -85,B 0,C 180,E1 1745.171,E2 1745.171} C_VEL
LIN {X 0,Y 166.029,Z 1192.839,A -85,B 0,C 180,E1 1738.019,E2 1738.019} C_VEL
LIN {X 0,Y 162.031,Z 1196.959,A -85,B 0,C 180,E1 1729.842,E2 1729.842} C_VEL
LIN {X 0,Y 160.176,Z 1200.002,A -85,B 0,C 180,E1 1720.795,E2 1720.795} C_VEL
LIN {X 0,Y 159.918,Z 1201.329,A -85,B 0,C 180,E1 1713.586,E2 1713.586} C_VEL
LIN {X 0,Y 159.914,Z 1201.71,A -85,B 0,C 180,E1 1707.493,E2 1707.493} C_VEL
LIN {X 0,Y 160.077,Z 1201.337,A -85,B 0,C 180,E1 1700.655,E2 1700.655} C_VEL
LIN {X 0,Y 161.634,Z 1199.649,A -85,B 0,C 180,E1 1691.611,E2 1691.611} C_VEL
LIN {X 0,Y 165.743,Z 1196.467,A -85,B 0,C 180,E1 1682.712,E2 1682.712} C_VEL
LIN {X 0,Y 171.952,Z 1192.44,A -85,B 0,C 180,E1 1675.076,E2 1675.076} C_VEL
LIN {X 0,Y 180.174,Z 1187.483,A -85,B 0,C 180,E1 1668.247,E2 1668.247} C_VEL
LIN {X 0,Y 191.222,Z 1180.977,A -85,B 0,C 180,E1 1661.608,E2 1661.608} C_VEL
LIN {X 0,Y 207.478,Z 1171.279,A -85,B 0,C 180,E1 1654.507,E2 1654.507} C_VEL
LIN {X 0,Y 222.775,Z 1161.664,A -85,B 0,C 180,E1 1649.459,E2 1649.459} C_VEL
LIN {X 0,Y 238.012,Z 1151.598,A -85,B 0,C 180,E1 1645.42,E2 1645.42} C_VEL
LIN {X 0,Y 253.579,Z 1140.674,A -85,B 0,C 180,E1 1641.999,E2 1641.999} C_VEL
LIN {X 0,Y 273.022,Z 1126.08,A -85,B 0,C 180,E1 1638.467,E2 1638.467} C_VEL
LIN {X 0,Y 291.744,Z 1110.493,A -85,B 0,C 180,E1 1635.627,E2 1635.627} C_VEL
LIN {X 0,Y 307.535,Z 1096.279,A -85,B 0,C 180,E1 1633.564,E2 1633.564} C_VEL
LIN {X 0,Y 322.95,Z 1081.265,A -85,B 0,C 180,E1 1631.791,E2 1631.791} C_VEL
LIN {X 0,Y 339.248,Z 1064.002,A -85,B 0,C 180,E1 1630.135,E2 1630.135} C_VEL
LIN {X 0,Y 357.847,Z 1042.055,A -85,B 0,C 180,E1 1628.463,E2 1628.463} C_VEL
LIN {X 0,Y 371.393,Z 1024.274,A -85,B 0,C 180,E1 1627.368,E2 1627.368} C_VEL
LIN {X 0,Y 384.022,Z 1006.053,A -85,B 0,C 180,E1 1626.428,E2 1626.428} C_VEL
LIN {X 0,Y 395.847,Z 987.221,A -85,B 0,C 180,E1 1625.618,E2 1625.618} C_VEL
LIN {X 0,Y 408.391,Z 964.925,A -85,B 0,C 180,E1 1624.823,E2 1624.823} C_VEL
LIN {X 0,Y 420.819,Z 939.217,A -85,B 0,C 180,E1 1624.088,E2 1624.088} C_VEL
LIN {X 0,Y 429.594,Z 918.22,A -85,B 0,C 180,E1 1623.603,E2 1623.603} C_VEL
LIN {X 0,Y 436.88,Z 898.151,A -85,B 0,C 180,E1 1623.219,E2 1623.219} C_VEL
LIN {X 0,Y 442.907,Z 878.838,A -85,B 0,C 180,E1 1622.907,E2 1622.907} C_VEL
LIN {X 0,Y 436.374,Z 899.617,A -85,B 0,C 180,E1 1622.553,E2 1622.553} C_VEL
LIN {X 0,Y 427.465,Z 923.639,A -85,B 0,C 180,E1 1622.05,E2 1622.05} C_VEL
LIN {X 0,Y 416.021,Z 949.435,A -85,B 0,C 180,E1 1621.377,E2 1621.377} C_VEL
LIN {X 0,Y 405.334,Z 970.293,A -85,B 0,C 180,E1 1620.707,E2 1620.707} C_VEL
LIN {X 0,Y 394.446,Z 989.248,A -85,B 0,C 180,E1 1619.983,E2 1619.983} C_VEL
LIN {X 0,Y 382.645,Z 1007.767,A -85,B 0,C 180,E1 1619.138,E2 1619.138} C_VEL
LIN {X 0,Y 366.695,Z 1030.278,A -85,B 0,C 180,E1 1617.905,E2 1617.905} C_VEL
LIN {X 0,Y 350.109,Z 1050.843,A -85,B 0,C 180,E1 1616.487,E2 1616.487} C_VEL
LIN {X 0,Y 335.681,Z 1067.154,A -85,B 0,C 180,E1 1615.11,E2 1615.11} C_VEL
LIN {X 0,Y 320.982,Z 1082.421,A -85,B 0,C 180,E1 1613.558,E2 1613.558} C_VEL
LIN {X 0,Y 303.48,Z 1099.129,A -85,B 0,C 180,E1 1611.474,E2 1611.474} C_VEL
LIN {X 0,Y 283.462,Z 1116.35,A -85,B 0,C 180,E1 1608.694,E2 1608.694} C_VEL
LIN {X 0,Y 267.754,Z 1128.749,A -85,B 0,C 180,E1 1606.144,E2 1606.144} C_VEL
LIN {X 0,Y 252.054,Z 1140.288,A -85,B 0,C 180,E1 1603.167,E2 1603.167} C_VEL
LIN {X 0,Y 236.662,Z 1150.875,A -85,B 0,C 180,E1 1599.704,E2 1599.704} C_VEL
LIN {X 0,Y 218.15,Z 1162.837,A -85,B 0,C 180,E1 1594.544,E2 1594.544} C_VEL
LIN {X 0,Y 201.789,Z 1172.571,A -85,B 0,C 180,E1 1588.648,E2 1588.648} C_VEL
LIN {X 0,Y 190.021,Z 1179.379,A -85,B 0,C 180,E1 1583.11,E2 1583.11} C_VEL
LIN {X 0,Y 179.761,Z 1185.243,A -85,B 0,C 180,E1 1576.772,E2 1576.772} C_VEL
LIN {X 0,Y 170.608,Z 1190.62,A -85,B 0,C 180,E1 1568.786,E2 1568.786} C_VEL
LIN {X 0,Y 163.898,Z 1194.831,A -85,B 0,C 180,E1 1559.211,E2 1559.211} C_VEL
LIN {X 0,Y 161.033,Z 1196.989,A -85,B 0,C 180,E1 1551.107,E2 1551.107} C_VEL
LIN {X 0,Y 160.089,Z 1197.973,A -85,B 0,C 180,E1 1544.097,E2 1544.097} C_VEL
LIN {X 0,Y 159.934,Z 1198.162,A -85,B 0,C 180,E1 1537.543,E2 1537.543} C_VEL
LIN {X 0,Y 159.951,Z 1197.642,A -85,B 0,C 180,E1 1531.073,E2 1531.073} C_VEL
LIN {X 0,Y 160.47,Z 1196.087,A -85,B 0,C 180,E1 1523.559,E2 1523.559} C_VEL
LIN {X 0,Y 162.558,Z 1193.245,A -85,B 0,C 180,E1 1515.392,E2 1515.392} C_VEL
LIN {X 0,Y 166.567,Z 1189.431,A -85,B 0,C 180,E1 1507.778,E2 1507.778} C_VEL
LIN {X 0,Y 172.384,Z 1184.754,A -85,B 0,C 180,E1 1500.84,E2 1500.84} C_VEL
LIN {X 0,Y 180.567,Z 1178.73,A -85,B 0,C 180,E1 1494.056,E2 1494.056} C_VEL
LIN {X 0,Y 192.265,Z 1170.482,A -85,B 0,C 180,E1 1487.056,E2 1487.056} C_VEL
LIN {X 0,Y 206.813,Z 1160.019,A -85,B 0,C 180,E1 1480.618,E2 1480.618} C_VEL
LIN {X 0,Y 220.753,Z 1149.676,A -85,B 0,C 180,E1 1475.828,E2 1475.828} C_VEL
LIN {X 0,Y 234.528,Z 1139.006,A -85,B 0,C 180,E1 1471.96,E2 1471.96} C_VEL
LIN {X 0,Y 251.465,Z 1125.15,A -85,B 0,C 180,E1 1468.026,E2 1468.026} C_VEL
LIN {X 0,Y 269.404,Z 1109.109,A -85,B 0,C 180,E1 1464.563,E2 1464.563} C_VEL
LIN {X 0,Y 284.304,Z 1094.722,A -85,B 0,C 180,E1 1462.106,E2 1462.106} C_VEL
LIN {X 0,Y 298.116,Z 1080.373,A -85,B 0,C 180,E1 1460.095,E2 1460.095} C_VEL
LIN {X 0,Y 312.633,Z 1064.083,A -85,B 0,C 180,E1 1458.216,E2 1458.216} C_VEL
LIN {X 0,Y 330.09,Z 1042.521,A -85,B 0,C 180,E1 1456.212,E2 1456.212} C_VEL
LIN {X 0,Y 344.312,Z 1022.845,A -85,B 0,C 180,E1 1454.753,E2 1454.753} C_VEL
LIN {X 0,Y 356.135,Z 1004.871,A -85,B 0,C 180,E1 1453.641,E2 1453.641} C_VEL
LIN {X 0,Y 367.377,Z 986.017,A -85,B 0,C 180,E1 1452.651,E2 1452.651} C_VEL
LIN {X 0,Y 380.236,Z 961.937,A -85,B 0,C 180,E1 1451.61,E2 1451.61} C_VEL
LIN {X 0,Y 391.386,Z 937.42,A -85,B 0,C 180,E1 1450.76,E2 1450.76} C_VEL
LIN {X 0,Y 399.722,Z 916.429,A -85,B 0,C 180,E1 1450.161,E2 1450.161} C_VEL
LIN {X 0,Y 406.971,Z 895.327,A -85,B 0,C 180,E1 1449.658,E2 1449.658} C_VEL
LIN {X 0,Y 414.594,Z 868.912,A -85,B 0,C 180,E1 1449.154,E2 1449.154} C_VEL
LIN {X 0,Y 420.497,Z 841.767,A -85,B 0,C 180,E1 1448.757,E2 1448.757} C_VEL
LIN {X 0,Y 424.143,Z 819.368,A -85,B 0,C 180,E1 1448.46,E2 1448.46} C_VEL
LIN {X 0,Y 441.273,Z 673.468,A -85,B 0,C 180,E1 1446.603,E2 1446.603} C_VEL
LIN {X 0,Y 440.84,Z 671.221,A -85,B 0,C 180,E1 1444.423,E2 1444.423} C_VEL
LIN {X 0,Y 440.884,Z 671.5,A -85,B 0,C 180,E1 1441.3,E2 1441.3} C_VEL
LIN {X 0,Y 441.263,Z 673.79,A -85,B 0,C 180,E1 1439.439,E2 1439.439} C_VEL
LIN {X 0,Y 434.767,Z 729.438,A -85,B 0,C 180,E1 1438.744,E2 1438.744} C_VEL
LIN {X 0,Y 433.797,Z 737.139,A -85,B 0,C 180,E1 1438.78,E2 1438.78} C_VEL
LIN {X 0,Y 430.957,Z 757.748,A -85,B 0,C 180,E1 1439.354,E2 1439.354} C_VEL
LIN {X 0,Y 430.134,Z 764.354,A -85,B 0,C 180,E1 1439.372,E2 1439.372} C_VEL
LIN {X 0,Y 422.711,Z 825.07,A -85,B 0,C 180,E1 1438.618,E2 1438.618} C_VEL
LIN {X 0,Y 417.066,Z 855.473,A -85,B 0,C 180,E1 1438.216,E2 1438.216} C_VEL
LIN {X 0,Y 411.323,Z 878.45,A -85,B 0,C 180,E1 1437.878,E2 1437.878} C_VEL
LIN {X 0,Y 404.842,Z 899.88,A -85,B 0,C 180,E1 1437.488,E2 1437.488} C_VEL
LIN {X 0,Y 396.625,Z 922.93,A -85,B 0,C 180,E1 1436.965,E2 1436.965} C_VEL
LIN {X 0,Y 385.298,Z 949.632,A -85,B 0,C 180,E1 1436.208,E2 1436.208} C_VEL
LIN {X 0,Y 375.123,Z 970.341,A -85,B 0,C 180,E1 1435.48,E2 1435.48} C_VEL
LIN {X 0,Y 364.534,Z 989.604,A -85,B 0,C 180,E1 1434.67,E2 1434.67} C_VEL
LIN {X 0,Y 353.075,Z 1008.408,A -85,B 0,C 180,E1 1433.724,E2 1433.724} C_VEL
LIN {X 0,Y 337.954,Z 1030.792,A -85,B 0,C 180,E1 1432.37,E2 1432.37} C_VEL
LIN {X 0,Y 321.646,Z 1052.014,A -85,B 0,C 180,E1 1430.75,E2 1430.75} C_VEL
LIN {X 0,Y 307.897,Z 1068.367,A -85,B 0,C 180,E1 1429.222,E2 1429.222} C_VEL
LIN {X 0,Y 293.945,Z 1083.68,A -85,B 0,C 180,E1 1427.491,E2 1427.491} C_VEL
LIN {X 0,Y 278.108,Z 1099.746,A -85,B 0,C 180,E1 1425.271,E2 1425.271} C_VEL
LIN {X 0,Y 258.533,Z 1117.812,A -85,B 0,C 180,E1 1422.067,E2 1422.067} C_VEL
LIN {X 0,Y 242.838,Z 1131.124,A -85,B 0,C 180,E1 1419.009,E2 1419.009} C_VEL
LIN {X 0,Y 228.279,Z 1142.718,A -85,B 0,C 180,E1 1415.653,E2 1415.653} C_VEL
LIN {X 0,Y 213.662,Z 1153.724,A -85,B 0,C 180,E1 1411.618,E2 1411.618} C_VEL
LIN {X 0,Y 196.371,Z 1166.095,A -85,B 0,C 180,E1 1405.577,E2 1405.577} C_VEL
LIN {X 0,Y 183.013,Z 1175.249,A -85,B 0,C 180,E1 1399.414,E2 1399.414} C_VEL
LIN {X 0,Y 172.696,Z 1182.35,A -85,B 0,C 180,E1 1393.096,E2 1393.096} C_VEL
LIN {X 0,Y 164.397,Z 1188.282,A -85,B 0,C 180,E1 1386.156,E2 1386.156} C_VEL
LIN {X 0,Y 157.572,Z 1193.726,A -85,B 0,C 180,E1 1377.597,E2 1377.597} C_VEL
LIN {X 0,Y 153.279,Z 1198.065,A -85,B 0,C 180,E1 1367.463,E2 1367.463} C_VEL
LIN {X 0,Y 152.079,Z 1200.237,A -85,B 0,C 180,E1 1359.462,E2 1359.462} C_VEL
LIN {X 0,Y 151.916,Z 1201.302,A -85,B 0,C 180,E1 1352.642,E2 1352.642} C_VEL
LIN {X 0,Y 151.914,Z 1201.655,A -85,B 0,C 180,E1 1346.605,E2 1346.605} C_VEL
LIN {X 0,Y 152.164,Z 1201.207,A -85,B 0,C 180,E1 1339.399,E2 1339.399} C_VEL
LIN {X 0,Y 154.136,Z 1199.372,A -85,B 0,C 180,E1 1329.892,E2 1329.892} C_VEL
LIN {X 0,Y 158.684,Z 1196.277,A -85,B 0,C 180,E1 1320.977,E2 1320.977} C_VEL
LIN {X 0,Y 165.394,Z 1192.317,A -85,B 0,C 180,E1 1313.24,E2 1313.24} C_VEL
LIN {X 0,Y 174.488,Z 1187.238,A -85,B 0,C 180,E1 1306.104,E2 1306.104} C_VEL
LIN {X 0,Y 186.327,Z 1180.704,A -85,B 0,C 180,E1 1299.402,E2 1299.402} C_VEL
LIN {X 0,Y 204.162,Z 1170.547,A -85,B 0,C 180,E1 1292.088,E2 1292.088} C_VEL
LIN {X 0,Y 219.506,Z 1161.303,A -85,B 0,C 180,E1 1287.348,E2 1287.348} C_VEL
LIN {X 0,Y 234.544,Z 1151.715,A -85,B 0,C 180,E1 1283.575,E2 1283.575} C_VEL
LIN {X 0,Y 250.451,Z 1140.904,A -85,B 0,C 180,E1 1280.253,E2 1280.253} C_VEL
LIN {X 0,Y 269.649,Z 1126.888,A -85,B 0,C 180,E1 1276.93,E2 1276.93} C_VEL
LIN {X 0,Y 289.624,Z 1110.718,A -85,B 0,C 180,E1 1274.05,E2 1274.05} C_VEL
LIN {X 0,Y 305.707,Z 1096.534,A -85,B 0,C 180,E1 1272.062,E2 1272.062} C_VEL
LIN {X 0,Y 321.207,Z 1081.717,A -85,B 0,C 180,E1 1270.374,E2 1270.374} C_VEL
LIN {X 0,Y 336.97,Z 1065.334,A -85,B 0,C 180,E1 1268.855,E2 1268.855} C_VEL
LIN {X 0,Y 355.523,Z 1044.013,A -85,B 0,C 180,E1 1267.271,E2 1267.271} C_VEL
LIN {X 0,Y 370.56,Z 1024.575,A -85,B 0,C 180,E1 1266.119,E2 1266.119} C_VEL
LIN {X 0,Y 383.531,Z 1006.078,A -85,B 0,C 180,E1 1265.208,E2 1265.208} C_VEL
LIN {X 0,Y 395.142,Z 987.797,A -85,B 0,C 180,E1 1264.458,E2 1264.458} C_VEL
LIN {X 0,Y 406.819,Z 967.345,A -85,B 0,C 180,E1 1263.758,E2 1263.758} C_VEL
LIN {X 0,Y 420.075,Z 940.617,A -85,B 0,C 180,E1 1263.018,E2 1263.018} C_VEL
LIN {X 0,Y 422.652,Z 934.778,A -85,B 0,C 180,E1 1262.878,E2 1262.878} C_VEL
LIN {X 0,Y 413.29,Z 954.721,A -85,B 0,C 180,E1 1262.346,E2 1262.346} C_VEL
LIN {X 0,Y 402.671,Z 974.766,A -85,B 0,C 180,E1 1261.708,E2 1261.708} C_VEL
LIN {X 0,Y 387.981,Z 999.194,A -85,B 0,C 180,E1 1260.762,E2 1260.762} C_VEL
LIN {X 0,Y 373.401,Z 1020.361,A -85,B 0,C 180,E1 1259.741,E2 1259.741} C_VEL
LIN {X 0,Y 360.534,Z 1037.283,A -85,B 0,C 180,E1 1258.758,E2 1258.758} C_VEL
LIN {X 0,Y 346.751,Z 1053.84,A -85,B 0,C 180,E1 1257.62,E2 1257.62} C_VEL
LIN {X 0,Y 330.703,Z 1071.448,A -85,B 0,C 180,E1 1256.144,E2 1256.144} C_VEL
LIN {X 0,Y 310.63,Z 1091.222,A -85,B 0,C 180,E1 1254.05,E2 1254.05} C_VEL
LIN {X 0,Y 293.801,Z 1106.215,A -85,B 0,C 180,E1 1252.024,E2 1252.024} C_VEL
LIN {X 0,Y 278.282,Z 1118.973,A -85,B 0,C 180,E1 1249.89,E2 1249.89} C_VEL
LIN {X 0,Y 262.315,Z 1131.134,A -85,B 0,C 180,E1 1247.366,E2 1247.366} C_VEL
LIN {X 0,Y 242.762,Z 1144.948,A -85,B 0,C 180,E1 1243.668,E2 1243.668} C_VEL
LIN {X 0,Y 223.572,Z 1157.17,A -85,B 0,C 180,E1 1239.178,E2 1239.178} C_VEL
LIN {X 0,Y 208.329,Z 1166.272,A -85,B 0,C 180,E1 1234.712,E2 1234.712} C_VEL
LIN {X 0,Y 194.6,Z 1174.051,A -85,B 0,C 180,E1 1229.676,E2 1229.676} C_VEL
LIN {X 0,Y 179.982,Z 1182.084,A -85,B 0,C 180,E1 1222.599,E2 1222.599} C_VEL
LIN {X 0,Y 167.804,Z 1188.517,A -85,B 0,C 180,E1 1214.197,E2 1214.197} C_VEL
LIN {X 0,Y 160.22,Z 1192.669,A -85,B 0,C 180,E1 1206.359,E2 1206.359} C_VEL
LIN {X 0,Y 155.598,Z 1195.433,A -85,B 0,C 180,E1 1198.811,E2 1198.811} C_VEL
LIN {X 0,Y 153.001,Z 1197.248,A -85,B 0,C 180,E1 1191.064,E2 1191.064} C_VEL
LIN {X 0,Y 152.112,Z 1198.073,A -85,B 0,C 180,E1 1184.463,E2 1184.463} C_VEL
LIN {X 0,Y 151.934,Z 1198.237,A -85,B 0,C 180,E1 1177.562,E2 1177.562} C_VEL
LIN {X 0,Y 151.959,Z 1197.693,A -85,B 0,C 180,E1 1170.753,E2 1170.753} C_VEL
LIN {X 0,Y 152.564,Z 1196.115,A -85,B 0,C 180,E1 1162.845,E2 1162.845} C_VEL
LIN {X 0,Y 154.932,Z 1193.25,A -85,B 0,C 180,E1 1154.272,E2 1154.272} C_VEL
LIN {X 0,Y 159.283,Z 1189.468,A -85,B 0,C 180,E1 1146.422,E2 1146.422} C_VEL
LIN {X 0,Y 165.689,Z 1184.71,A -85,B 0,C 180,E1 1139.138,E2 1139.138} C_VEL
LIN {X 0,Y 174.485,Z 1178.662,A -85,B 0,C 180,E1 1132.18,E2 1132.18} C_VEL
LIN {X 0,Y 187.857,Z 1169.791,A -85,B 0,C 180,E1 1124.635,E2 1124.635} C_VEL
LIN {X 0,Y 202.864,Z 1159.411,A -85,B 0,C 180,E1 1118.392,E2 1118.392} C_VEL
LIN {X 0,Y 216.771,Z 1149.494,A -85,B 0,C 180,E1 1113.872,E2 1113.872} C_VEL
LIN {X 0,Y 231.055,Z 1138.791,A -85,B 0,C 180,E1 1110.06,E2 1110.06} C_VEL
LIN {X 0,Y 249.309,Z 1124.272,A -85,B 0,C 180,E1 1106.054,E2 1106.054} C_VEL
LIN {X 0,Y 267.718,Z 1108.071,A -85,B 0,C 180,E1 1102.704,E2 1102.704} C_VEL
LIN {X 0,Y 281.833,Z 1094.714,A -85,B 0,C 180,E1 1100.509,E2 1100.509} C_VEL
LIN {X 0,Y 296.559,Z 1079.681,A -85,B 0,C 180,E1 1098.478,E2 1098.478} C_VEL
LIN {X 0,Y 313.288,Z 1061.13,A -85,B 0,C 180,E1 1096.449,E2 1096.449} C_VEL
LIN {X 0,Y 330.173,Z 1040.152,A -85,B 0,C 180,E1 1094.633,E2 1094.633} C_VEL
LIN {X 0,Y 343.263,Z 1022.199,A -85,B 0,C 180,E1 1093.369,E2 1093.369} C_VEL
LIN {X 0,Y 355.134,Z 1004.333,A -85,B 0,C 180,E1 1092.317,E2 1092.317} C_VEL
LIN {X 0,Y 367.101,Z 984.411,A -85,B 0,C 180,E1 1091.321,E2 1091.321} C_VEL
LIN {X 0,Y 381.043,Z 957.96,A -85,B 0,C 180,E1 1090.255,E2 1090.255} C_VEL
LIN {X 0,Y 390.828,Z 936.473,A -85,B 0,C 180,E1 1089.556,E2 1089.556} C_VEL
LIN {X 0,Y 398.873,Z 916.338,A -85,B 0,C 180,E1 1089.008,E2 1089.008} C_VEL
LIN {X 0,Y 406.193,Z 895.197,A -85,B 0,C 180,E1 1088.527,E2 1088.527} C_VEL
LIN {X 0,Y 413.855,Z 868.834,A -85,B 0,C 180,E1 1088.047,E2 1088.047} C_VEL
LIN {X 0,Y 419.764,Z 841.886,A -85,B 0,C 180,E1 1087.669,E2 1087.669} C_VEL
LIN {X 0,Y 423.458,Z 819.455,A -85,B 0,C 180,E1 1087.379,E2 1087.379} C_VEL
LIN {X 0,Y 440.026,Z 680.456,A -85,B 0,C 180,E1 1085.656,E2 1085.656} C_VEL
LIN {X 0,Y 439.844,Z 679.15,A -85,B 0,C 180,E1 1084.302,E2 1084.302} C_VEL
LIN {X 0,Y 439.886,Z 679.374,A -85,B 0,C 180,E1 1081.433,E2 1081.433} C_VEL
LIN {X 0,Y 440.005,Z 680.776,A -85,B 0,C 180,E1 1080.396,E2 1080.396} C_VEL
LIN {X 0,Y 430.134,Z 764.354,A -85,B 0,C 180,E1 1079.372,E2 1079.372} C_VEL
LIN {X 0,Y 429.167,Z 772.057,A -85,B 0,C 180,E1 1079.411,E2 1079.411} C_VEL
LIN {X 0,Y 426.374,Z 792.662,A -85,B 0,C 180,E1 1080.002,E2 1080.002} C_VEL
LIN {X 0,Y 425.553,Z 799.269,A -85,B 0,C 180,E1 1080.02,E2 1080.02} C_VEL
LIN {X 0,Y 420.512,Z 835.207,A -85,B 0,C 180,E1 1079.576,E2 1079.576} C_VEL
LIN {X 0,Y 415.672,Z 858.85,A -85,B 0,C 180,E1 1079.271,E2 1079.271} C_VEL
LIN {X 0,Y 410.05,Z 880.65,A -85,B 0,C 180,E1 1078.96,E2 1078.96} C_VEL
LIN {X 0,Y 402.833,Z 903.832,A -85,B 0,C 180,E1 1078.545,E2 1078.545} C_VEL
LIN {X 0,Y 392.217,Z 931.843,A -85,B 0,C 180,E1 1077.903,E2 1077.903} C_VEL
LIN {X 0,Y 382.895,Z 952.764,A -85,B 0,C 180,E1 1077.306,E2 1077.306} C_VEL
LIN {X 0,Y 373.098,Z 972.26,A -85,B 0,C 180,E1 1076.638,E2 1076.638} C_VEL
LIN {X 0,Y 361.919,Z 992.16,A -85,B 0,C 180,E1 1075.823,E2 1075.823} C_VEL
LIN {X 0,Y 347.46,Z 1015.156,A -85,B 0,C 180,E1 1074.673,E2 1074.673} C_VEL
LIN {X 0,Y 332.199,Z 1036.423,A -85,B 0,C 180,E1 1073.346,E2 1073.346} C_VEL
LIN {X 0,Y 318.845,Z 1053.355,A -85,B 0,C 180,E1 1072.069,E2 1072.069} C_VEL
LIN {X 0,Y 304.555,Z 1069.971,A -85,B 0,C 180,E1 1070.552,E2 1070.552} C_VEL
LIN {X 0,Y 286.812,Z 1088.885,A -85,B 0,C 180,E1 1068.414,E2 1068.414} C_VEL
LIN {X 0,Y 268.153,Z 1106.664,A -85,B 0,C 180,E1 1065.81,E2 1065.81} C_VEL
LIN {X 0,Y 252.654,Z 1120.298,A -85,B 0,C 180,E1 1063.28,E2 1063.28} C_VEL
LIN {X 0,Y 237.693,Z 1132.557,A -85,B 0,C 180,E1 1060.439,E2 1060.439} C_VEL
LIN {X 0,Y 221.042,Z 1145.326,A -85,B 0,C 180,E1 1056.675,E2 1056.675} C_VEL
LIN {X 0,Y 201.885,Z 1158.917,A -85,B 0,C 180,E1 1051.24,E2 1051.24} C_VEL
LIN {X 0,Y 187.869,Z 1168.332,A -85,B 0,C 180,E1 1046.128,E2 1046.128} C_VEL
LIN {X 0,Y 175.958,Z 1176.102,A -85,B 0,C 180,E1 1040.609,E2 1040.609} C_VEL
LIN {X 0,Y 164.795,Z 1183.38,A -85,B 0,C 180,E1 1033.765,E2 1033.765} C_VEL
LIN {X 0,Y 153.935,Z 1190.8,A -85,B 0,C 180,E1 1023.961,E2 1023.961} C_VEL
LIN {X 0,Y 148.064,Z 1195.347,A -85,B 0,C 180,E1 1015.18,E2 1015.18} C_VEL
LIN {X 0,Y 145.181,Z 1198.282,A -85,B 0,C 180,E1 1007.228,E2 1007.228} C_VEL
LIN {X 0,Y 144.084,Z 1200.192,A -85,B 0,C 180,E1 999.589,E2 999.589} C_VEL
LIN {X 0,Y 143.916,Z 1201.206,A -85,B 0,C 180,E1 992.789,E2 992.789} C_VEL
LIN {X 0,Y 143.914,Z 1201.561,A -85,B 0,C 180,E1 986.417,E2 986.417} C_VEL
LIN {X 0,Y 144.213,Z 1201.127,A -85,B 0,C 180,E1 978.808,E2 978.808} C_VEL
LIN {X 0,Y 146.459,Z 1199.326,A -85,B 0,C 180,E1 968.789,E2 968.789} C_VEL
LIN {X 0,Y 151.494,Z 1196.248,A -85,B 0,C 180,E1 959.457,E2 959.457} C_VEL
LIN {X 0,Y 159.031,Z 1192.182,A -85,B 0,C 180,E1 951.228,E2 951.228} C_VEL
LIN {X 0,Y 169.052,Z 1186.993,A -85,B 0,C 180,E1 943.817,E2 943.817} C_VEL
LIN {X 0,Y 182.922,Z 1179.827,A -85,B 0,C 180,E1 936.535,E2 936.535} C_VEL
LIN {X 0,Y 201.232,Z 1169.814,A -85,B 0,C 180,E1 929.598,E2 929.598} C_VEL
LIN {X 0,Y 216.8,Z 1160.787,A -85,B 0,C 180,E1 925.107,E2 925.107} C_VEL
LIN {X 0,Y 232.929,Z 1150.817,A -85,B 0,C 180,E1 921.333,E2 921.333} C_VEL
LIN {X 0,Y 250.207,Z 1139.347,A -85,B 0,C 180,E1 917.996,E2 917.996} C_VEL
LIN {X 0,Y 272.728,Z 1122.912,A -85,B 0,C 180,E1 914.436,E2 914.436} C_VEL
LIN {X 0,Y 290.429,Z 1108.66,A -85,B 0,C 180,E1 912.115,E2 912.115} C_VEL
LIN {X 0,Y 305.932,Z 1095.123,A -85,B 0,C 180,E1 910.346,E2 910.346} C_VEL
LIN {X 0,Y 322.636,Z 1079.274,A -85,B 0,C 180,E1 908.663,E2 908.663} C_VEL
LIN {X 0,Y 342.446,Z 1058.464,A -85,B 0,C 180,E1 906.919,E2 906.919} C_VEL
LIN {X 0,Y 358.215,Z 1039.89,A -85,B 0,C 180,E1 905.689,E2 905.689} C_VEL
LIN {X 0,Y 371.721,Z 1022.406,A -85,B 0,C 180,E1 904.741,E2 904.741} C_VEL
LIN {X 0,Y 384.344,Z 1004.423,A -85,B 0,C 180,E1 903.915,E2 903.915} C_VEL
LIN {X 0,Y 397.047,Z 984.381,A -85,B 0,C 180,E1 903.155,E2 903.155} C_VEL
LIN {X 0,Y 402.282,Z 975.37,A -85,B 0,C 180,E1 902.849,E2 902.849} C_VEL
LIN {X 0,Y 386.661,Z 1000.889,A -85,B 0,C 180,E1 901.903,E2 901.903} C_VEL
LIN {X 0,Y 373.005,Z 1020.476,A -85,B 0,C 180,E1 900.999,E2 900.999} C_VEL
LIN {X 0,Y 359.95,Z 1037.457,A -85,B 0,C 180,E1 900.064,E2 900.064} C_VEL
LIN {X 0,Y 345.511,Z 1054.572,A -85,B 0,C 180,E1 898.939,E2 898.939} C_VEL
LIN {X 0,Y 327.306,Z 1074.19,A -85,B 0,C 180,E1 897.345,E2 897.345} C_VEL
LIN {X 0,Y 307.94,Z 1092.652,A -85,B 0,C 180,E1 895.42,E2 895.42} C_VEL
LIN {X 0,Y 291.792,Z 1106.738,A -85,B 0,C 180,E1 893.575,E2 893.575} C_VEL
LIN {X 0,Y 275.978,Z 1119.456,A -85,B 0,C 180,E1 891.52,E2 891.52} C_VEL
LIN {X 0,Y 258.165,Z 1132.669,A -85,B 0,C 180,E1 888.834,E2 888.834} C_VEL
LIN {X 0,Y 236.081,Z 1147.531,A -85,B 0,C 180,E1 884.776,E2 884.776} C_VEL
LIN {X 0,Y 219.039,Z 1157.979,A -85,B 0,C 180,E1 880.891,E2 880.891} C_VEL
LIN {X 0,Y 203.635,Z 1166.801,A -85,B 0,C 180,E1 876.564,E2 876.564} C_VEL
LIN {X 0,Y 188.235,Z 1175.119,A -85,B 0,C 180,E1 871.093,E2 871.093} C_VEL
LIN {X 0,Y 171.524,Z 1183.65,A -85,B 0,C 180,E1 862.996,E2 862.996} C_VEL
LIN {X 0,Y 160.367,Z 1189.171,A -85,B 0,C 180,E1 855.206,E2 855.206} C_VEL
LIN {X 0,Y 152.795,Z 1193.005,A -85,B 0,C 180,E1 847.485,E2 847.485} C_VEL
LIN {X 0,Y 147.618,Z 1195.832,A -85,B 0,C 180,E1 839.098,E2 839.098} C_VEL
LIN {X 0,Y 144.887,Z 1197.574,A -85,B 0,C 180,E1 830.605,E2 830.605} C_VEL
LIN {X 0,Y 144.038,Z 1198.258,A -85,B 0,C 180,E1 823.241,E2 823.241} C_VEL
LIN {X 0,Y 143.923,Z 1198.289,A -85,B 0,C 180,E1 817.182,E2 817.182} C_VEL
LIN {X 0,Y 143.97,Z 1197.744,A -85,B 0,C 180,E1 810.396,E2 810.396} C_VEL
LIN {X 0,Y 144.613,Z 1196.254,A -85,B 0,C 180,E1 802.45,E2 802.45} C_VEL
LIN {X 0,Y 147.189,Z 1193.41,A -85,B 0,C 180,E1 793.421,E2 793.421} C_VEL
LIN {X 0,Y 151.972,Z 1189.594,A -85,B 0,C 180,E1 785.096,E2 785.096} C_VEL
LIN {X 0,Y 159.005,Z 1184.76,A -85,B 0,C 180,E1 777.422,E2 777.422} C_VEL
LIN {X 0,Y 168.599,Z 1178.592,A -85,B 0,C 180,E1 770.17,E2 770.17} C_VEL
LIN {X 0,Y 182.972,Z 1169.549,A -85,B 0,C 180,E1 762.46,E2 762.46} C_VEL
LIN {X 0,Y 198.551,Z 1159.266,A -85,B 0,C 180,E1 756.317,E2 756.317} C_VEL
LIN {X 0,Y 213.051,Z 1149.31,A -85,B 0,C 180,E1 751.846,E2 751.846} C_VEL
LIN {X 0,Y 228.603,Z 1138.014,A -85,B 0,C 180,E1 747.929,E2 747.929} C_VEL
LIN {X 0,Y 248.247,Z 1122.624,A -85,B 0,C 180,E1 743.892,E2 743.892} C_VEL
LIN {X 0,Y 265.339,Z 1107.908,A -85,B 0,C 180,E1 740.977,E2 740.977} C_VEL
LIN {X 0,Y 279.956,Z 1094.342,A -85,B 0,C 180,E1 738.832,E2 738.832} C_VEL
LIN {X 0,Y 293.832,Z 1080.447,A -85,B 0,C 180,E1 737.017,E2 737.017} C_VEL
LIN {X 0,Y 308.863,Z 1064.145,A -85,B 0,C 180,E1 735.265,E2 735.265} C_VEL
LIN {X 0,Y 326.874,Z 1042.556,A -85,B 0,C 180,E1 733.409,E2 733.409} C_VEL
LIN {X 0,Y 341.499,Z 1022.863,A -85,B 0,C 180,E1 732.06,E2 732.06} C_VEL
LIN {X 0,Y 353.515,Z 1005.053,A -85,B 0,C 180,E1 731.051,E2 731.051} C_VEL
LIN {X 0,Y 365.151,Z 985.993,A -85,B 0,C 180,E1 730.13,E2 730.13} C_VEL
LIN {X 0,Y 378.298,Z 961.852,A -85,B 0,C 180,E1 729.176,E2 729.176} C_VEL
LIN {X 0,Y 389.636,Z 937.391,A -85,B 0,C 180,E1 728.402,E2 728.402} C_VEL
LIN {X 0,Y 397.71,Z 917.493,A -85,B 0,C 180,E1 727.881,E2 727.881} C_VEL
LIN {X 0,Y 404.857,Z 897.238,A -85,B 0,C 180,E1 727.436,E2 727.436} C_VEL
LIN {X 0,Y 411.489,Z 875.134,A -85,B 0,C 180,E1 727.037,E2 727.037} C_VEL
LIN {X 0,Y 418.196,Z 847.276,A -85,B 0,C 180,E1 726.643,E2 726.643} C_VEL
LIN {X 0,Y 422.63,Z 821.619,A -85,B 0,C 180,E1 726.322,E2 726.322} C_VEL
LIN {X 0,Y 438.908,Z 687.378,A -85,B 0,C 180,E1 724.704,E2 724.704} C_VEL
LIN {X 0,Y 438.844,Z 687.092,A -85,B 0,C 180,E1 721.959,E2 721.959} C_VEL
LIN {X 0,Y 438.888,Z 687.615,A -85,B 0,C 180,E1 721.36,E2 721.36} C_VEL
LIN {X 0,Y 425.553,Z 799.269,A -85,B 0,C 180,E1 720.02,E2 720.02} C_VEL
LIN {X 0,Y 424.592,Z 806.967,A -85,B 0,C 180,E1 720.057,E2 720.057} C_VEL
LIN {X 0,Y 421.506,Z 827.519,A -85,B 0,C 180,E1 720.66,E2 720.66} C_VEL
LIN {X 0,Y 420.316,Z 834.073,A -85,B 0,C 180,E1 720.683,E2 720.683} C_VEL
LIN {X 0,Y 415.338,Z 858.331,A -85,B 0,C 180,E1 720.383,E2 720.383} C_VEL
LIN {X 0,Y 409.702,Z 880.103,A -85,B 0,C 180,E1 720.089,E2 720.089} C_VEL
LIN {X 0,Y 402.766,Z 902.324,A -85,B 0,C 180,E1 719.716,E2 719.716} C_VEL
LIN {X 0,Y 392.37,Z 929.952,A -85,B 0,C 180,E1 719.124,E2 719.124} C_VEL
LIN {X 0,Y 382.58,Z 951.862,A -85,B 0,C 180,E1 718.538,E2 718.538} C_VEL
LIN {X 0,Y 372.818,Z 971.198,A -85,B 0,C 180,E1 717.914,E2 717.914} C_VEL
LIN {X 0,Y 361.899,Z 990.555,A -85,B 0,C 180,E1 717.168,E2 717.168} C_VEL
LIN {X 0,Y 349.702,Z 1010.008,A -85,B 0,C 180,E1 716.266,E2 716.266} C_VEL
LIN {X 0,Y 332.893,Z 1033.813,A -85,B 0,C 180,E1 714.913,E2 714.913} C_VEL
LIN {X 0,Y 317.959,Z 1052.612,A -85,B 0,C 180,E1 713.577,E2 713.577} C_VEL
LIN {X 0,Y 303.802,Z 1068.897,A -85,B 0,C 180,E1 712.165,E2 712.165} C_VEL
LIN {X 0,Y 288.925,Z 1084.62,A -85,B 0,C 180,E1 710.507,E2 710.507} C_VEL
LIN {X 0,Y 269.805,Z 1103.098,A -85,B 0,C 180,E1 708.063,E2 708.063} C_VEL
LIN {X 0,Y 251.229,Z 1119.196,A -85,B 0,C 180,E1 705.271,E2 705.271} C_VEL
LIN {X 0,Y 235.84,Z 1131.551,A -85,B 0,C 180,E1 702.541,E2 702.541} C_VEL
LIN {X 0,Y 220.139,Z 1143.306,A -85,B 0,C 180,E1 699.25,E2 699.25} C_VEL
LIN {X 0,Y 201.379,Z 1156.453,A -85,B 0,C 180,E1 694.407,E2 694.407} C_VEL
LIN {X 0,Y 183.953,Z 1167.659,A -85,B 0,C 180,E1 688.582,E2 688.582} C_VEL
LIN {X 0,Y 170.739,Z 1175.868,A -85,B 0,C 180,E1 682.793,E2 682.793} C_VEL
LIN {X 0,Y 159.329,Z 1182.856,A -85,B 0,C 180,E1 676.196,E2 676.196} C_VEL
LIN {X 0,Y 148.153,Z 1189.981,A -85,B 0,C 180,E1 666.919,E2 666.919} C_VEL
LIN {X 0,Y 140.631,Z 1195.194,A -85,B 0,C 180,E1 656.612,E2 656.612} C_VEL
LIN {X 0,Y 137.396,Z 1198.149,A -85,B 0,C 180,E1 648.237,E2 648.237} C_VEL
LIN {X 0,Y 136.116,Z 1200.079,A -85,B 0,C 180,E1 640.15,E2 640.15} C_VEL
LIN {X 0,Y 135.916,Z 1201.11,A -85,B 0,C 180,E1 632.953,E2 632.953} C_VEL
LIN {X 0,Y 135.914,Z 1201.443,A -85,B 0,C 180,E1 626.628,E2 626.628} C_VEL
LIN {X 0,Y 136.229,Z 1201.072,A -85,B 0,C 180,E1 618.572,E2 618.572} C_VEL
LIN {X 0,Y 138.671,Z 1199.395,A -85,B 0,C 180,E1 607.981,E2 607.981} C_VEL
LIN {X 0,Y 144.631,Z 1196.106,A -85,B 0,C 180,E1 597.505,E2 597.505} C_VEL
LIN {X 0,Y 152.783,Z 1192.091,A -85,B 0,C 180,E1 589.125,E2 589.125} C_VEL
LIN {X 0,Y 163.367,Z 1187.004,A -85,B 0,C 180,E1 581.698,E2 581.698} C_VEL
LIN {X 0,Y 177.415,Z 1180.16,A -85,B 0,C 180,E1 574.634,E2 574.634} C_VEL
LIN {X 0,Y 196.5,Z 1170.29,A -85,B 0,C 180,E1 567.704,E2 567.704} C_VEL
LIN {X 0,Y 213.106,Z 1161.042,A -85,B 0,C 180,E1 563.133,E2 563.133} C_VEL
LIN {X 0,Y 229.191,Z 1151.448,A -85,B 0,C 180,E1 559.557,E2 559.557} C_VEL
LIN {X 0,Y 246.034,Z 1140.627,A -85,B 0,C 180,E1 556.448,E2 556.448} C_VEL
LIN {X 0,Y 265.284,Z 1127.228,A -85,B 0,C 180,E1 553.492,E2 553.492} C_VEL
LIN {X 0,Y 286.972,Z 1110.411,A -85,B 0,C 180,E1 550.723,E2 550.723} C_VEL
LIN {X 0,Y 303.797,Z 1096.069,A -85,B 0,C 180,E1 548.899,E2 548.899} C_VEL
LIN {X 0,Y 319.607,Z 1081.398,A -85,B 0,C 180,E1 547.385,E2 547.385} C_VEL
LIN {X 0,Y 335.799,Z 1065,A -85,B 0,C 180,E1 546.01,E2 546.01} C_VEL
LIN {X 0,Y 355.078,Z 1043.301,A -85,B 0,C 180,E1 544.566,E2 544.566} C_VEL
LIN {X 0,Y 370.103,Z 1024.264,A -85,B 0,C 180,E1 543.563,E2 543.563} C_VEL
LIN {X 0,Y 381.793,Z 1008.013,A -85,B 0,C 180,E1 542.825,E2 542.825} C_VEL
LIN {X 0,Y 365.627,Z 1030.18,A -85,B 0,C 180,E1 541.788,E2 541.788} C_VEL
LIN {X 0,Y 348.281,Z 1050.989,A -85,B 0,C 180,E1 540.554,E2 540.554} C_VEL
LIN {X 0,Y 333.426,Z 1067.163,A -85,B 0,C 180,E1 539.378,E2 539.378} C_VEL
LIN {X 0,Y 318.141,Z 1082.389,A -85,B 0,C 180,E1 538.045,E2 538.045} C_VEL
LIN {X 0,Y 300.58,Z 1098.394,A -85,B 0,C 180,E1 536.314,E2 536.314} C_VEL
LIN {X 0,Y 278.599,Z 1116.371,A -85,B 0,C 180,E1 533.784,E2 533.784} C_VEL
LIN {X 0,Y 260.911,Z 1129.439,A -85,B 0,C 180,E1 531.379,E2 531.379} C_VEL
LIN {X 0,Y 243.749,Z 1141.105,A -85,B 0,C 180,E1 528.63,E2 528.63} C_VEL
LIN {X 0,Y 224.68,Z 1153.048,A -85,B 0,C 180,E1 524.945,E2 524.945} C_VEL
LIN {X 0,Y 203.534,Z 1165.008,A -85,B 0,C 180,E1 519.765,E2 519.765} C_VEL
LIN {X 0,Y 187.791,Z 1173.215,A -85,B 0,C 180,E1 514.788,E2 514.788} C_VEL
LIN {X 0,Y 173.703,Z 1180.146,A -85,B 0,C 180,E1 509.054,E2 509.054} C_VEL
LIN {X 0,Y 160.403,Z 1186.441,A -85,B 0,C 180,E1 501.758,E2 501.758} C_VEL
LIN {X 0,Y 147.646,Z 1192.323,A -85,B 0,C 180,E1 491.26,E2 491.26} C_VEL
LIN {X 0,Y 140.987,Z 1195.51,A -85,B 0,C 180,E1 482.132,E2 482.132} C_VEL
LIN {X 0,Y 137.534,Z 1197.367,A -85,B 0,C 180,E1 473.567,E2 473.567} C_VEL
LIN {X 0,Y 136.209,Z 1198.253,A -85,B 0,C 180,E1 465.758,E2 465.758} C_VEL
LIN {X 0,Y 135.935,Z 1198.435,A -85,B 0,C 180,E1 458.458,E2 458.458} C_VEL
LIN {X 0,Y 135.947,Z 1197.998,A -85,B 0,C 180,E1 451.263,E2 451.263} C_VEL
LIN {X 0,Y 136.541,Z 1196.616,A -85,B 0,C 180,E1 442.847,E2 442.847} C_VEL
LIN {X 0,Y 139.479,Z 1193.571,A -85,B 0,C 180,E1 432.476,E2 432.476} C_VEL
LIN {X 0,Y 144.666,Z 1189.776,A -85,B 0,C 180,E1 423.745,E2 423.745} C_VEL
LIN {X 0,Y 151.97,Z 1185.119,A -85,B 0,C 180,E1 415.994,E2 415.994} C_VEL
LIN {X 0,Y 161.423,Z 1179.411,A -85,B 0,C 180,E1 408.959,E2 408.959} C_VEL
LIN {X 0,Y 173.371,Z 1172.266,A -85,B 0,C 180,E1 402.419,E2 402.419} C_VEL
LIN {X 0,Y 190.422,Z 1161.807,A -85,B 0,C 180,E1 395.521,E2 395.521} C_VEL
LIN {X 0,Y 207.382,Z 1150.637,A -85,B 0,C 180,E1 390.339,E2 390.339} C_VEL
LIN {X 0,Y 222.553,Z 1140.043,A -85,B 0,C 180,E1 386.611,E2 386.611} C_VEL
LIN {X 0,Y 238.501,Z 1128.129,A -85,B 0,C 180,E1 383.345,E2 383.345} C_VEL
LIN {X 0,Y 257.632,Z 1112.697,A -85,B 0,C 180,E1 380.079,E2 380.079} C_VEL
LIN {X 0,Y 275.7,Z 1096.456,A -85,B 0,C 180,E1 377.479,E2 377.479} C_VEL
LIN {X 0,Y 290.678,Z 1081.846,A -85,B 0,C 180,E1 375.601,E2 375.601} C_VEL
LIN {X 0,Y 305.48,Z 1066.164,A -85,B 0,C 180,E1 373.953,E2 373.953} C_VEL
LIN {X 0,Y 321.017,Z 1048.184,A -85,B 0,C 180,E1 372.411,E2 372.411} C_VEL
LIN {X 0,Y 338.521,Z 1025.492,A -85,B 0,C 180,E1 370.857,E2 370.857} C_VEL
LIN {X 0,Y 351.554,Z 1006.559,A -85,B 0,C 180,E1 369.814,E2 369.814} C_VEL
LIN {X 0,Y 362.719,Z 988.638,A -85,B 0,C 180,E1 368.973,E2 368.973} C_VEL
LIN {X 0,Y 373.305,Z 969.817,A -85,B 0,C 180,E1 368.234,E2 368.234} C_VEL
LIN {X 0,Y 384.257,Z 947.97,A -85,B 0,C 180,E1 367.516,E2 367.516} C_VEL
LIN {X 0,Y 395.743,Z 921.171,A -85,B 0,C 180,E1 366.806,E2 366.806} C_VEL
LIN {X 0,Y 403.67,Z 899.28,A -85,B 0,C 180,E1 366.338,E2 366.338} C_VEL
LIN {X 0,Y 410.204,Z 878.045,A -85,B 0,C 180,E1 365.965,E2 365.965} C_VEL
LIN {X 0,Y 415.904,Z 855.678,A -85,B 0,C 180,E1 365.649,E2 365.649} C_VEL
LIN {X 0,Y 421.494,Z 826.951,A -85,B 0,C 180,E1 365.298,E2 365.298} C_VEL
LIN {X 0,Y 427.715,Z 778.38,A -85,B 0,C 180,E1 364.724,E2 364.724} C_VEL
LIN {X 0,Y 437.821,Z 695.02,A -85,B 0,C 180,E1 363.732,E2 363.732} C_VEL
LIN {X 0,Y 437.807,Z 695.181,A -85,B 0,C 180,E1 362.32,E2 362.32} C_VEL
LIN {X 0,Y 422.141,Z 822.545,A -85,B 0,C 180,E1 360.824,E2 360.824} C_VEL
LIN {X 0,Y 420.316,Z 834.073,A -85,B 0,C 180,E1 360.683,E2 360.683} C_VEL
LIN {X 0,Y 418.852,Z 841.683,A -85,B 0,C 180,E1 360.743,E2 360.743} C_VEL
LIN {X 0,Y 414.767,Z 859.796,A -85,B 0,C 180,E1 361.314,E2 361.314} C_VEL
LIN {X 0,Y 412.901,Z 867.336,A -85,B 0,C 180,E1 361.378,E2 361.378} C_VEL
LIN {X 0,Y 412.643,Z 868.416,A -85,B 0,C 180,E1 361.368,E2 361.368} C_VEL
LIN {X 0,Y 404.787,Z 895.063,A -85,B 0,C 180,E1 360.981,E2 360.981} C_VEL
LIN {X 0,Y 397.425,Z 915.927,A -85,B 0,C 180,E1 360.6,E2 360.6} C_VEL
LIN {X 0,Y 388.956,Z 936.68,A -85,B 0,C 180,E1 360.142,E2 360.142} C_VEL
LIN {X 0,Y 378.966,Z 958.105,A -85,B 0,C 180,E1 359.566,E2 359.566} C_VEL
LIN {X 0,Y 364.555,Z 984.805,A -85,B 0,C 180,E1 358.673,E2 358.673} C_VEL
LIN {X 0,Y 352.209,Z 1004.788,A -85,B 0,C 180,E1 357.84,E2 357.84} C_VEL
LIN {X 0,Y 340.21,Z 1022.345,A -85,B 0,C 180,E1 356.967,E2 356.967} C_VEL
LIN {X 0,Y 327.284,Z 1039.576,A -85,B 0,C 180,E1 355.939,E2 355.939} C_VEL
LIN {X 0,Y 311.85,Z 1058.302,A -85,B 0,C 180,E1 354.596,E2 354.596} C_VEL
LIN {X 0,Y 292.356,Z 1079.407,A -85,B 0,C 180,E1 352.67,E2 352.67} C_VEL
LIN {X 0,Y 276.154,Z 1095.246,A -85,B 0,C 180,E1 350.833,E2 350.833} C_VEL
LIN {X 0,Y 259.984,Z 1109.779,A -85,B 0,C 180,E1 348.731,E2 348.731} C_VEL
LIN {X 0,Y 240.389,Z 1125.977,A -85,B 0,C 180,E1 345.732,E2 345.732} C_VEL
LIN {X 0,Y 220.639,Z 1140.6,A -85,B 0,C 180,E1 342.051,E2 342.051} C_VEL
LIN {X 0,Y 205.198,Z 1151.23,A -85,B 0,C 180,E1 338.545,E2 338.545} C_VEL
LIN {X 0,Y 189.806,Z 1161.178,A -85,B 0,C 180,E1 334.267,E2 334.267} C_VEL
LIN {X 0,Y 172.865,Z 1171.557,A -85,B 0,C 180,E1 328.24,E2 328.24} C_VEL
LIN {X 0,Y 156.762,Z 1180.857,A -85,B 0,C 180,E1 320.369,E2 320.369} C_VEL
LIN {X 0,Y 145.787,Z 1187.184,A -85,B 0,C 180,E1 312.766,E2 312.766} C_VEL
LIN {X 0,Y 137.588,Z 1192.152,A -85,B 0,C 180,E1 304.532,E2 304.532} C_VEL
LIN {X 0,Y 131.977,Z 1196.009,A -85,B 0,C 180,E1 295.634,E2 295.634} C_VEL
LIN {X 0,Y 128.98,Z 1198.715,A -85,B 0,C 180,E1 286.67,E2 286.67} C_VEL
LIN {X 0,Y 128.025,Z 1200.312,A -85,B 0,C 180,E1 278.535,E2 278.535} C_VEL
LIN {X 0,Y 127.918,Z 1201.082,A -85,B 0,C 180,E1 271.793,E2 271.793} C_VEL
LIN {X 0,Y 127.93,Z 1201.358,A -85,B 0,C 180,E1 264.62,E2 264.62} C_VEL
LIN {X 0,Y 128.589,Z 1200.804,A -85,B 0,C 180,E1 255.594,E2 255.594} C_VEL
LIN {X 0,Y 131.851,Z 1198.888,A -85,B 0,C 180,E1 244.872,E2 244.872} C_VEL
LIN {X 0,Y 138.137,Z 1195.871,A -85,B 0,C 180,E1 235.124,E2 235.124} C_VEL
LIN {X 0,Y 147.037,Z 1191.875,A -85,B 0,C 180,E1 226.624,E2 226.624} C_VEL
LIN {X 0,Y 158.495,Z 1186.761,A -85,B 0,C 180,E1 219.111,E2 219.111} C_VEL
LIN {X 0,Y 174.796,Z 1179.285,A -85,B 0,C 180,E1 211.538,E2 211.538} C_VEL
LIN {X 0,Y 194.255,Z 1169.562,A -85,B 0,C 180,E1 205.057,E2 205.057} C_VEL
LIN {X 0,Y 210.759,Z 1160.686,A -85,B 0,C 180,E1 200.84,E2 200.84} C_VEL
LIN {X 0,Y 228.222,Z 1150.55,A -85,B 0,C 180,E1 197.24,E2 197.24} C_VEL
LIN {X 0,Y 247.327,Z 1138.502,A -85,B 0,C 180,E1 194.015,E2 194.015} C_VEL
LIN {X 0,Y 270.051,Z 1122.567,A -85,B 0,C 180,E1 190.885,E2 190.885} C_VEL
LIN {X 0,Y 287.411,Z 1109.124,A -85,B 0,C 180,E1 188.888,E2 188.888} C_VEL
LIN {X 0,Y 303.407,Z 1095.651,A -85,B 0,C 180,E1 187.285,E2 187.285} C_VEL
LIN {X 0,Y 319.616,Z 1080.781,A -85,B 0,C 180,E1 185.843,E2 185.843} C_VEL
LIN {X 0,Y 336.982,Z 1063.333,A -85,B 0,C 180,E1 184.477,E2 184.477} C_VEL
LIN {X 0,Y 356.481,Z 1041.319,A -85,B 0,C 180,E1 183.126,E2 183.126} C_VEL
LIN {X 0,Y 361.333,Z 1035.388,A -85,B 0,C 180,E1 182.813,E2 182.813} C_VEL
LIN {X 0,Y 346.655,Z 1052.609,A -85,B 0,C 180,E1 181.818,E2 181.818} C_VEL
LIN {X 0,Y 331.98,Z 1068.306,A -85,B 0,C 180,E1 180.724,E2 180.724} C_VEL
LIN {X 0,Y 315.281,Z 1084.613,A -85,B 0,C 180,E1 179.346,E2 179.346} C_VEL
LIN {X 0,Y 293.296,Z 1103.874,A -85,B 0,C 180,E1 177.253,E2 177.253} C_VEL
LIN {X 0,Y 274.849,Z 1118.341,A -85,B 0,C 180,E1 175.2,E2 175.2} C_VEL
LIN {X 0,Y 257.884,Z 1130.531,A -85,B 0,C 180,E1 173.004,E2 173.004} C_VEL
LIN {X 0,Y 240.373,Z 1142.098,A -85,B 0,C 180,E1 170.342,E2 170.342} C_VEL
LIN {X 0,Y 219.116,Z 1154.949,A -85,B 0,C 180,E1 166.396,E2 166.396} C_VEL
LIN {X 0,Y 199.073,Z 1165.734,A -85,B 0,C 180,E1 161.67,E2 161.67} C_VEL
LIN {X 0,Y 183.107,Z 1173.695,A -85,B 0,C 180,E1 156.848,E2 156.848} C_VEL
LIN {X 0,Y 168.071,Z 1180.709,A -85,B 0,C 180,E1 150.986,E2 150.986} C_VEL
LIN {X 0,Y 152.144,Z 1187.792,A -85,B 0,C 180,E1 142.324,E2 142.324} C_VEL
LIN {X 0,Y 140.365,Z 1192.721,A -85,B 0,C 180,E1 132.586,E2 132.586} C_VEL
LIN {X 0,Y 133.613,Z 1195.662,A -85,B 0,C 180,E1 123.624,E2 123.624} C_VEL
LIN {X 0,Y 129.764,Z 1197.493,A -85,B 0,C 180,E1 114.586,E2 114.586} C_VEL
LIN {X 0,Y 128.255,Z 1198.353,A -85,B 0,C 180,E1 106.298,E2 106.298} C_VEL
LIN {X 0,Y 127.935,Z 1198.51,A -85,B 0,C 180,E1 98.538,E2 98.538} C_VEL
LIN {X 0,Y 127.945,Z 1198.116,A -85,B 0,C 180,E1 91.342,E2 91.342} C_VEL
LIN {X 0,Y 128.592,Z 1196.755,A -85,B 0,C 180,E1 82.402,E2 82.402} C_VEL
LIN {X 0,Y 131.811,Z 1193.731,A -85,B 0,C 180,E1 71.42,E2 71.42} C_VEL
LIN {X 0,Y 137.448,Z 1189.958,A -85,B 0,C 180,E1 62.251,E2 62.251} C_VEL
LIN {X 0,Y 145.735,Z 1185.074,A -85,B 0,C 180,E1 53.838,E2 53.838} C_VEL
LIN {X 0,Y 156.434,Z 1179.044,A -85,B 0,C 180,E1 46.344,E2 46.344} C_VEL
LIN {X 0,Y 171.099,Z 1170.787,A -85,B 0,C 180,E1 38.99,E2 38.99} C_VEL
LIN {X 0,Y 189.345,Z 1159.855,A -85,B 0,C 180,E1 32.335,E2 32.335} C_VEL
LIN {X 0,Y 204.909,Z 1149.948,A -85,B 0,C 180,E1 27.966,E2 27.966} C_VEL
LIN {X 0,Y 220.719,Z 1139.198,A -85,B 0,C 180,E1 24.346,E2 24.346} C_VEL
LIN {X 0,Y 240.426,Z 1124.763,A -85,B 0,C 180,E1 20.653,E2 20.653} C_VEL
LIN {X 0,Y 260.155,Z 1108.593,A -85,B 0,C 180,E1 17.604,E2 17.604} C_VEL
LIN {X 0,Y 276.04,Z 1094.428,A -85,B 0,C 180,E1 15.523,E2 15.523} C_VEL
LIN {X 0,Y 290.421,Z 1080.52,A -85,B 0,C 180,E1 13.858,E2 13.858} C_VEL
LIN {X 0,Y 305.935,Z 1064.205,A -85,B 0,C 180,E1 12.253,E2 12.253} C_VEL
LIN {X 0,Y 324.923,Z 1041.989,A -85,B 0,C 180,E1 10.519,E2 10.519} C_VEL
LIN {X 0,Y 339.452,Z 1022.866,A -85,B 0,C 180,E1 9.331,E2 9.331} C_VEL
LIN {X 0,Y 351.749,Z 1005.026,A -85,B 0,C 180,E1 8.418,E2 8.418} C_VEL
LIN {X 0,Y 363.636,Z 985.937,A -85,B 0,C 180,E1 7.584,E2 7.584} C_VEL
LIN {X 0,Y 377.049,Z 961.729,A -85,B 0,C 180,E1 6.722,E2 6.722} C_VEL
LIN {X 0,Y 388.119,Z 938.336,A -85,B 0,C 180,E1 6.053,E2 6.053} C_VEL
LIN {X 0,Y 396.333,Z 918.54,A -85,B 0,C 180,E1 5.582,E2 5.582} C_VEL
LIN {X 0,Y 403.843,Z 897.688,A -85,B 0,C 180,E1 5.166,E2 5.166} C_VEL
LIN {X 0,Y 410.522,Z 875.841,A -85,B 0,C 180,E1 4.81,E2 4.81} C_VEL
LIN {X 0,Y 417.277,Z 848.559,A -85,B 0,C 180,E1 4.459,E2 4.459} C_VEL
LIN {X 0,Y 421.978,Z 822,A -85,B 0,C 180,E1 4.15,E2 4.15} C_VEL
LIN {X 0,Y 434.096,Z 725.087,A -85,B 0,C 180,E1 3.029,E2 3.029} C_VEL
LIN {X 0,Y 421.851,Z 822.949,A -85,B 0,C 180,E1 1.908,E2 1.908} C_VEL
LIN {X 0,Y 416.859,Z 850.664,A -85,B 0,C 180,E1 1.581,E2 1.581} C_VEL
LIN {X 0,Y 412.643,Z 868.416,A -85,B 0,C 180,E1 1.368,E2 1.368} C_VEL
LIN {X 0,Y 410.677,Z 875.924,A -85,B 0,C 180,E1 1.411,E2 1.411} C_VEL
LIN {X 0,Y 404.707,Z 894.701,A -85,B 0,C 180,E1 1.986,E2 1.986} C_VEL
LIN {X 0,Y 402.219,Z 902.045,A -85,B 0,C 180,E1 2.009,E2 2.009} C_VEL
LIN {X 0,Y 392.089,Z 928.728,A -85,B 0,C 180,E1 1.504,E2 1.504} C_VEL
LIN {X 0,Y 381.508,Z 952.041,A -85,B 0,C 180,E1 0.951,E2 0.951} C_VEL
LIN {X 0,Y 371.237,Z 971.965,A -85,B 0,C 180,E1 0.375,E2 0.375} C_VEL
LIN {X 0,Y 359.963,Z 991.487,A -85,B 0,C 180,E1 -0.302,E2 -0.302} C_VEL
LIN {X 0,Y 345.047,Z 1014.559,A -85,B 0,C 180,E1 -1.284,E2 -1.284} C_VEL
LIN {X 0,Y 329.254,Z 1035.858,A -85,B 0,C 180,E1 -2.411,E2 -2.411} C_VEL
LIN {X 0,Y 314.94,Z 1053.341,A -85,B 0,C 180,E1 -3.547,E2 -3.547} C_VEL
LIN {X 0,Y 300.046,Z 1069.939,A -85,B 0,C 180,E1 -4.864,E2 -4.864} C_VEL
LIN {X 0,Y 281.403,Z 1088.877,A -85,B 0,C 180,E1 -6.734,E2 -6.734} C_VEL
LIN {X 0,Y 261.863,Z 1106.478,A -85,B 0,C 180,E1 -9.007,E2 -9.007} C_VEL
LIN {X 0,Y 245.662,Z 1119.861,A -85,B 0,C 180,E1 -11.212,E2 -11.212} C_VEL
LIN {X 0,Y 229.566,Z 1132.135,A -85,B 0,C 180,E1 -13.762,E2 -13.762} C_VEL
LIN {X 0,Y 211.437,Z 1144.922,A -85,B 0,C 180,E1 -17.203,E2 -17.203} C_VEL
LIN {X 0,Y 190.188,Z 1158.543,A -85,B 0,C 180,E1 -22.286,E2 -22.286} C_VEL
LIN {X 0,Y 174.273,Z 1167.973,A -85,B 0,C 180,E1 -27.213,E2 -27.213} C_VEL
LIN {X 0,Y 159.955,Z 1176.031,A -85,B 0,C 180,E1 -32.946,E2 -32.946} C_VEL
LIN {X 0,Y 145.963,Z 1183.671,A -85,B 0,C 180,E1 -40.501,E2 -40.501} C_VEL
LIN {X 0,Y 132.705,Z 1190.917,A -85,B 0,C 180,E1 -51.289,E2 -51.289} C_VEL
LIN {X 0,Y 125.537,Z 1195.216,A -85,B 0,C 180,E1 -60.93,E2 -60.93} C_VEL
LIN {X 0,Y 121.676,Z 1198.115,A -85,B 0,C 180,E1 -70.309,E2 -70.309} C_VEL
LIN {X 0,Y 120.135,Z 1199.988,A -85,B 0,C 180,E1 -79.448,E2 -79.448} C_VEL
LIN {X 0,Y 119.915,Z 1200.94,A -85,B 0,C 180,E1 -87.13,E2 -87.13} C_VEL
LIN {X 0,Y 119.917,Z 1201.271,A -85,B 0,C 180,E1 -94.302,E2 -94.302} C_VEL
LIN {X 0,Y 120.376,Z 1200.911,A -85,B 0,C 180,E1 -102.958,E2 -102.958} C_VEL
LIN {X 0,Y 123.579,Z 1199.304,A -85,B 0,C 180,E1 -114.879,E2 -114.879} C_VEL
LIN {X 0,Y 131.039,Z 1196.005,A -85,B 0,C 180,E1 -126.522,E2 -126.522} C_VEL
LIN {X 0,Y 141.084,Z 1191.867,A -85,B 0,C 180,E1 -135.706,E2 -135.706} C_VEL
LIN {X 0,Y 153.349,Z 1186.772,A -85,B 0,C 180,E1 -143.318,E2 -143.318} C_VEL
LIN {X 0,Y 169.848,Z 1179.621,A -85,B 0,C 180,E1 -150.602,E2 -150.602} C_VEL
LIN {X 0,Y 190.849,Z 1169.639,A -85,B 0,C 180,E1 -157.229,E2 -157.229} C_VEL
LIN {X 0,Y 208.76,Z 1160.329,A -85,B 0,C 180,E1 -161.499,E2 -161.499} C_VEL
LIN {X 0,Y 226.57,Z 1150.27,A -85,B 0,C 180,E1 -164.908,E2 -164.908} C_VEL
LIN {X 0,Y 248.159,Z 1136.949,A -85,B 0,C 180,E1 -168.257,E2 -168.257} C_VEL
LIN {X 0,Y 270.258,Z 1121.547,A -85,B 0,C 180,E1 -171.042,E2 -171.042} C_VEL
LIN {X 0,Y 288.146,Z 1107.837,A -85,B 0,C 180,E1 -172.937,E2 -172.937} C_VEL
LIN {X 0,Y 305.356,Z 1093.414,A -85,B 0,C 180,E1 -174.515,E2 -174.515} C_VEL
LIN {X 0,Y 324.722,Z 1075.597,A -85,B 0,C 180,E1 -176.06,E2 -176.06} C_VEL
LIN {X 0,Y 340.778,Z 1059.124,A -85,B 0,C 180,E1 -177.206,E2 -177.206} C_VEL
LIN {X 0,Y 320.688,Z 1079.253,A -85,B 0,C 180,E1 -178.673,E2 -178.673} C_VEL
LIN {X 0,Y 303.958,Z 1094.381,A -85,B 0,C 180,E1 -180.067,E2 -180.067} C_VEL
LIN {X 0,Y 287.696,Z 1107.838,A -85,B 0,C 180,E1 -181.593,E2 -181.593} C_VEL
LIN {X 0,Y 269.48,Z 1121.63,A -85,B 0,C 180,E1 -183.555,E2 -183.555} C_VEL
LIN {X 0,Y 246.457,Z 1137.325,A -85,B 0,C 180,E1 -186.523,E2 -186.523} C_VEL
LIN {X 0,Y 227.124,Z 1149.097,A -85,B 0,C 180,E1 -189.563,E2 -189.563} C_VEL
LIN {X 0,Y 209.318,Z 1159.018,A -85,B 0,C 180,E1 -192.979,E2 -192.979} C_VEL
LIN {X 0,Y 192.365,Z 1167.692,A -85,B 0,C 180,E1 -196.987,E2 -196.987} C_VEL
LIN {X 0,Y 172.713,Z 1176.976,A -85,B 0,C 180,E1 -203.007,E2 -203.007} C_VEL
LIN {X 0,Y 154.585,Z 1184.621,A -85,B 0,C 180,E1 -210.73,E2 -210.73} C_VEL
LIN {X 0,Y 142.164,Z 1189.603,A -85,B 0,C 180,E1 -218.239,E2 -218.239} C_VEL
LIN {X 0,Y 132.509,Z 1193.378,A -85,B 0,C 180,E1 -226.636,E2 -226.636} C_VEL
LIN {X 0,Y 125.524,Z 1196.151,A -85,B 0,C 180,E1 -236.113,E2 -236.113} C_VEL
LIN {X 0,Y 121.49,Z 1197.885,A -85,B 0,C 180,E1 -246.219,E2 -246.219} C_VEL
LIN {X 0,Y 120.101,Z 1198.559,A -85,B 0,C 180,E1 -255.539,E2 -255.539} C_VEL
LIN {X 0,Y 119.924,Z 1198.513,A -85,B 0,C 180,E1 -262.836,E2 -262.836} C_VEL
LIN {X 0,Y 120.007,Z 1197.963,A -85,B 0,C 180,E1 -270.479,E2 -270.479} C_VEL
LIN {X 0,Y 121.093,Z 1196.335,A -85,B 0,C 180,E1 -280.468,E2 -280.468} C_VEL
LIN {X 0,Y 124.642,Z 1193.578,A -85,B 0,C 180,E1 -290.671,E2 -290.671} C_VEL
LIN {X 0,Y 130.68,Z 1189.938,A -85,B 0,C 180,E1 -299.826,E2 -299.826} C_VEL
LIN {X 0,Y 139.255,Z 1185.277,A -85,B 0,C 180,E1 -308.135,E2 -308.135} C_VEL
LIN {X 0,Y 150.078,Z 1179.565,A -85,B 0,C 180,E1 -315.471,E2 -315.471} C_VEL
LIN {X 0,Y 163.461,Z 1172.415,A -85,B 0,C 180,E1 -322.102,E2 -322.102} C_VEL
LIN {X 0,Y 182.158,Z 1161.945,A -85,B 0,C 180,E1 -328.905,E2 -328.905} C_VEL
LIN {X 0,Y 200.422,Z 1150.767,A -85,B 0,C 180,E1 -333.897,E2 -333.897} C_VEL
LIN {X 0,Y 216.565,Z 1140.163,A -85,B 0,C 180,E1 -337.43,E2 -337.43} C_VEL
LIN {X 0,Y 233.383,Z 1128.241,A -85,B 0,C 180,E1 -340.484,E2 -340.484} C_VEL
LIN {X 0,Y 253.395,Z 1112.793,A -85,B 0,C 180,E1 -343.51,E2 -343.51} C_VEL
LIN {X 0,Y 273.077,Z 1095.713,A -85,B 0,C 180,E1 -346.004,E2 -346.004} C_VEL
LIN {X 0,Y 288.593,Z 1081.011,A -85,B 0,C 180,E1 -347.7,E2 -347.7} C_VEL
LIN {X 0,Y 303.874,Z 1065.209,A -85,B 0,C 180,E1 -349.19,E2 -349.19} C_VEL
LIN {X 0,Y 322.139,Z 1044.38,A -85,B 0,C 180,E1 -350.765,E2 -350.765} C_VEL
LIN {X 0,Y 338.325,Z 1023.405,A -85,B 0,C 180,E1 -352.015,E2 -352.015} C_VEL
LIN {X 0,Y 350.667,Z 1005.73,A -85,B 0,C 180,E1 -352.875,E2 -352.875} C_VEL
LIN {X 0,Y 362.19,Z 987.495,A -85,B 0,C 180,E1 -353.635,E2 -353.635} C_VEL
LIN {X 0,Y 374.262,Z 966.186,A -85,B 0,C 180,E1 -354.37,E2 -354.37} C_VEL
LIN {X 0,Y 387.362,Z 939.364,A -85,B 0,C 180,E1 -355.114,E2 -355.114} C_VEL
LIN {X 0,Y 396.129,Z 918.433,A -85,B 0,C 180,E1 -355.586,E2 -355.586} C_VEL
LIN {X 0,Y 403.697,Z 897.55,A -85,B 0,C 180,E1 -355.978,E2 -355.978} C_VEL
LIN {X 0,Y 410.579,Z 875.128,A -85,B 0,C 180,E1 -356.321,E2 -356.321} C_VEL
LIN {X 0,Y 417.533,Z 846.659,A -85,B 0,C 180,E1 -356.664,E2 -356.664} C_VEL
LIN {X 0,Y 421.948,Z 821.729,A -85,B 0,C 180,E1 -356.944,E2 -356.944} C_VEL
LIN {X 0,Y 422.197,Z 820.023,A -85,B 0,C 180,E1 -356.969,E2 -356.969} C_VEL
LIN {X 0,Y 418.301,Z 842.691,A -85,B 0,C 180,E1 -357.227,E2 -357.227} C_VEL
LIN {X 0,Y 411.987,Z 870.288,A -85,B 0,C 180,E1 -357.541,E2 -357.541} C_VEL
LIN {X 0,Y 404.453,Z 895.394,A -85,B 0,C 180,E1 -357.886,E2 -357.886} C_VEL
LIN {X 0,Y 402.219,Z 902.045,A -85,B 0,C 180,E1 -357.991,E2 -357.991} C_VEL
LIN {X 0,Y 399.635,Z 909.427,A -85,B 0,C 180,E1 -357.972,E2 -357.972} C_VEL
LIN {X 0,Y 392.314,Z 927.923,A -85,B 0,C 180,E1 -357.445,E2 -357.445} C_VEL
LIN {X 0,Y 389.228,Z 934.864,A -85,B 0,C 180,E1 -357.444,E2 -357.444} C_VEL
LIN {X 0,Y 379.707,Z 955.205,A -85,B 0,C 180,E1 -357.915,E2 -357.915} C_VEL
LIN {X 0,Y 368.078,Z 977.132,A -85,B 0,C 180,E1 -358.532,E2 -358.532} C_VEL
LIN {X 0,Y 352.978,Z 1001.862,A -85,B 0,C 180,E1 -359.399,E2 -359.399} C_VEL
LIN {X 0,Y 339.409,Z 1021.478,A -85,B 0,C 180,E1 -360.255,E2 -360.255} C_VEL
LIN {X 0,Y 326.457,Z 1038.446,A -85,B 0,C 180,E1 -361.143,E2 -361.143} C_VEL
LIN {X 0,Y 311.705,Z 1056.037,A -85,B 0,C 180,E1 -362.251,E2 -362.251} C_VEL
LIN {X 0,Y 292.634,Z 1076.547,A -85,B 0,C 180,E1 -363.871,E2 -363.871} C_VEL
LIN {X 0,Y 274.306,Z 1094.058,A -85,B 0,C 180,E1 -365.659,E2 -365.659} C_VEL
LIN {X 0,Y 258.166,Z 1108.164,A -85,B 0,C 180,E1 -367.475,E2 -367.475} C_VEL
LIN {X 0,Y 242.313,Z 1120.909,A -85,B 0,C 180,E1 -369.524,E2 -369.524} C_VEL
LIN {X 0,Y 225.004,Z 1133.728,A -85,B 0,C 180,E1 -372.135,E2 -372.135} C_VEL
LIN {X 0,Y 202.191,Z 1149.031,A -85,B 0,C 180,E1 -376.385,E2 -376.385} C_VEL
LIN {X 0,Y 184.706,Z 1159.669,A -85,B 0,C 180,E1 -380.524,E2 -380.524} C_VEL
LIN {X 0,Y 168.983,Z 1168.585,A -85,B 0,C 180,E1 -385.216,E2 -385.216} C_VEL
LIN {X 0,Y 153.994,Z 1176.608,A -85,B 0,C 180,E1 -391.008,E2 -391.008} C_VEL
LIN {X 0,Y 137.223,Z 1185.228,A -85,B 0,C 180,E1 -400.083,E2 -400.083} C_VEL
LIN {X 0,Y 125.197,Z 1191.299,A -85,B 0,C 180,E1 -410.059,E2 -410.059} C_VEL
LIN {X 0,Y 118.093,Z 1195.226,A -85,B 0,C 180,E1 -419.466,E2 -419.466} C_VEL
LIN {X 0,Y 113.85,Z 1198.098,A -85,B 0,C 180,E1 -429.431,E2 -429.431} C_VEL
LIN {X 0,Y 112.187,Z 1199.873,A -85,B 0,C 180,E1 -438.69,E2 -438.69} C_VEL
LIN {X 0,Y 111.915,Z 1200.844,A -85,B 0,C 180,E1 -446.925,E2 -446.925} C_VEL
LIN {X 0,Y 111.916,Z 1201.153,A -85,B 0,C 180,E1 -454.097,E2 -454.097} C_VEL
LIN {X 0,Y 112.351,Z 1200.881,A -85,B 0,C 180,E1 -462.853,E2 -462.853} C_VEL
LIN {X 0,Y 115.184,Z 1199.599,A -85,B 0,C 180,E1 -474.288,E2 -474.288} C_VEL
LIN {X 0,Y 123.664,Z 1196.3,A -85,B 0,C 180,E1 -487.913,E2 -487.913} C_VEL
LIN {X 0,Y 134.844,Z 1192.067,A -85,B 0,C 180,E1 -497.857,E2 -497.857} C_VEL
LIN {X 0,Y 147.849,Z 1187.04,A -85,B 0,C 180,E1 -505.592,E2 -505.592} C_VEL
LIN {X 0,Y 162.95,Z 1180.864,A -85,B 0,C 180,E1 -512.076,E2 -512.076} C_VEL
LIN {X 0,Y 183.712,Z 1171.724,A -85,B 0,C 180,E1 -518.539,E2 -518.539} C_VEL
LIN {X 0,Y 205.393,Z 1160.883,A -85,B 0,C 180,E1 -523.535,E2 -523.535} C_VEL
LIN {X 0,Y 223.608,Z 1150.924,A -85,B 0,C 180,E1 -526.818,E2 -526.818} C_VEL
LIN {X 0,Y 241.984,Z 1139.937,A -85,B 0,C 180,E1 -529.545,E2 -529.545} C_VEL
LIN {X 0,Y 264.363,Z 1125.213,A -85,B 0,C 180,E1 -532.273,E2 -532.273} C_VEL
LIN {X 0,Y 285.324,Z 1109.592,A -85,B 0,C 180,E1 -534.395,E2 -534.395} C_VEL
LIN {X 0,Y 302.733,Z 1095.346,A -85,B 0,C 180,E1 -535.899,E2 -535.899} C_VEL
LIN {X 0,Y 318.814,Z 1080.958,A -85,B 0,C 180,E1 -537.124,E2 -537.124} C_VEL
LIN {X 0,Y 320.029,Z 1079.827,A -85,B 0,C 180,E1 -537.225,E2 -537.225} C_VEL
LIN {X 0,Y 303.056,Z 1094.957,A -85,B 0,C 180,E1 -538.54,E2 -538.54} C_VEL
LIN {X 0,Y 285.96,Z 1108.86,A -85,B 0,C 180,E1 -540.036,E2 -540.036} C_VEL
LIN {X 0,Y 264.17,Z 1124.968,A -85,B 0,C 180,E1 -542.27,E2 -542.27} C_VEL
LIN {X 0,Y 242.222,Z 1139.229,A -85,B 0,C 180,E1 -544.973,E2 -544.973} C_VEL
LIN {X 0,Y 223.957,Z 1150.014,A -85,B 0,C 180,E1 -547.697,E2 -547.697} C_VEL
LIN {X 0,Y 205.747,Z 1159.829,A -85,B 0,C 180,E1 -550.995,E2 -550.995} C_VEL
LIN {X 0,Y 184.93,Z 1170.059,A -85,B 0,C 180,E1 -555.765,E2 -555.765} C_VEL
LIN {X 0,Y 163.984,Z 1179.135,A -85,B 0,C 180,E1 -562.213,E2 -562.213} C_VEL
LIN {X 0,Y 148.381,Z 1185.34,A -85,B 0,C 180,E1 -568.838,E2 -568.838} C_VEL
LIN {X 0,Y 134.914,Z 1190.362,A -85,B 0,C 180,E1 -576.834,E2 -576.834} C_VEL
LIN {X 0,Y 122.67,Z 1194.829,A -85,B 0,C 180,E1 -588.061,E2 -588.061} C_VEL
LIN {X 0,Y 115.096,Z 1197.481,A -85,B 0,C 180,E1 -600.892,E2 -600.892} C_VEL
LIN {X 0,Y 112.502,Z 1198.513,A -85,B 0,C 180,E1 -611.342,E2 -611.342} C_VEL
LIN {X 0,Y 111.941,Z 1198.707,A -85,B 0,C 180,E1 -620.231,E2 -620.231} C_VEL
LIN {X 0,Y 111.932,Z 1198.359,A -85,B 0,C 180,E1 -627.954,E2 -627.954} C_VEL
LIN {X 0,Y 112.496,Z 1197.211,A -85,B 0,C 180,E1 -637.15,E2 -637.15} C_VEL
LIN {X 0,Y 115.968,Z 1194.519,A -85,B 0,C 180,E1 -649.651,E2 -649.651} C_VEL
LIN {X 0,Y 123.34,Z 1190.32,A -85,B 0,C 180,E1 -661.255,E2 -661.255} C_VEL
LIN {X 0,Y 132.954,Z 1185.479,A -85,B 0,C 180,E1 -670.3,E2 -670.3} C_VEL
LIN {X 0,Y 144.795,Z 1179.635,A -85,B 0,C 180,E1 -677.945,E2 -677.945} C_VEL
LIN {X 0,Y 159.258,Z 1172.316,A -85,B 0,C 180,E1 -684.707,E2 -684.707} C_VEL
LIN {X 0,Y 179.605,Z 1161.337,A -85,B 0,C 180,E1 -691.596,E2 -691.596} C_VEL
LIN {X 0,Y 197.778,Z 1150.578,A -85,B 0,C 180,E1 -696.216,E2 -696.216} C_VEL
LIN {X 0,Y 214.414,Z 1139.942,A -85,B 0,C 180,E1 -699.609,E2 -699.609} C_VEL
LIN {X 0,Y 231.664,Z 1127.986,A -85,B 0,C 180,E1 -702.528,E2 -702.528} C_VEL
LIN {X 0,Y 253.006,Z 1111.709,A -85,B 0,C 180,E1 -705.523,E2 -705.523} C_VEL
LIN {X 0,Y 271.23,Z 1096.17,A -85,B 0,C 180,E1 -707.666,E2 -707.666} C_VEL
LIN {X 0,Y 286.98,Z 1081.493,A -85,B 0,C 180,E1 -709.276,E2 -709.276} C_VEL
LIN {X 0,Y 302.244,Z 1065.96,A -85,B 0,C 180,E1 -710.671,E2 -710.671} C_VEL
LIN {X 0,Y 319.746,Z 1046.386,A -85,B 0,C 180,E1 -712.091,E2 -712.091} C_VEL
LIN {X 0,Y 336.744,Z 1024.82,A -85,B 0,C 180,E1 -713.325,E2 -713.325} C_VEL
LIN {X 0,Y 349.765,Z 1006.433,A -85,B 0,C 180,E1 -714.175,E2 -714.175} C_VEL
LIN {X 0,Y 361.393,Z 988.261,A -85,B 0,C 180,E1 -714.893,E2 -714.893} C_VEL
LIN {X 0,Y 372.688,Z 968.616,A -85,B 0,C 180,E1 -715.538,E2 -715.538} C_VEL
LIN {X 0,Y 385.299,Z 943.722,A -85,B 0,C 180,E1 -716.208,E2 -716.208} C_VEL
LIN {X 0,Y 395.598,Z 919.587,A -85,B 0,C 180,E1 -716.729,E2 -716.729} C_VEL
LIN {X 0,Y 399.987,Z 908.315,A -85,B 0,C 180,E1 -716.946,E2 -716.946} C_VEL
LIN {X 0,Y 389.851,Z 933.45,A -85,B 0,C 180,E1 -717.414,E2 -717.414} C_VEL
LIN {X 0,Y 389.228,Z 934.864,A -85,B 0,C 180,E1 -717.444,E2 -717.444} C_VEL
LIN {X 0,Y 385.219,Z 943.943,A -85,B 0,C 180,E1 -717.489,E2 -717.489} C_VEL
LIN {X 0,Y 374.035,Z 966.119,A -85,B 0,C 180,E1 -717.118,E2 -717.118} C_VEL
LIN {X 0,Y 369.423,Z 974.4,A -85,B 0,C 180,E1 -717.193,E2 -717.193} C_VEL
LIN {X 0,Y 355.187,Z 998.15,A -85,B 0,C 180,E1 -717.946,E2 -717.946} C_VEL
LIN {X 0,Y 340.029,Z 1020.069,A -85,B 0,C 180,E1 -718.821,E2 -718.821} C_VEL
LIN {X 0,Y 326.468,Z 1037.749,A -85,B 0,C 180,E1 -719.674,E2 -719.674} C_VEL
LIN {X 0,Y 311.986,Z 1054.905,A -85,B 0,C 180,E1 -720.678,E2 -720.678} C_VEL
LIN {X 0,Y 294.158,Z 1074.073,A -85,B 0,C 180,E1 -722.069,E2 -722.069} C_VEL
LIN {X 0,Y 274.578,Z 1092.74,A -85,B 0,C 180,E1 -723.816,E2 -723.816} C_VEL
LIN {X 0,Y 257.206,Z 1107.744,A -85,B 0,C 180,E1 -725.617,E2 -725.617} C_VEL
LIN {X 0,Y 241.06,Z 1120.524,A -85,B 0,C 180,E1 -727.544,E2 -727.544} C_VEL
LIN {X 0,Y 222.461,Z 1134.02,A -85,B 0,C 180,E1 -730.156,E2 -730.156} C_VEL
LIN {X 0,Y 198.994,Z 1149.31,A -85,B 0,C 180,E1 -734.253,E2 -734.253} C_VEL
LIN {X 0,Y 181.077,Z 1159.855,A -85,B 0,C 180,E1 -738.237,E2 -738.237} C_VEL
LIN {X 0,Y 164.569,Z 1168.849,A -85,B 0,C 180,E1 -742.883,E2 -742.883} C_VEL
LIN {X 0,Y 147.568,Z 1177.517,A -85,B 0,C 180,E1 -749.2,E2 -749.2} C_VEL
LIN {X 0,Y 129.618,Z 1186.078,A -85,B 0,C 180,E1 -758.818,E2 -758.818} C_VEL
LIN {X 0,Y 118.299,Z 1191.417,A -85,B 0,C 180,E1 -768.107,E2 -768.107} C_VEL
LIN {X 0,Y 110.737,Z 1195.236,A -85,B 0,C 180,E1 -777.808,E2 -777.808} C_VEL
LIN {X 0,Y 106.052,Z 1198.08,A -85,B 0,C 180,E1 -788.424,E2 -788.424} C_VEL
LIN {X 0,Y 104.206,Z 1199.828,A -85,B 0,C 180,E1 -798.373,E2 -798.373} C_VEL
LIN {X 0,Y 103.915,Z 1200.771,A -85,B 0,C 180,E1 -807.24,E2 -807.24} C_VEL
LIN {X 0,Y 103.924,Z 1201.078,A -85,B 0,C 180,E1 -814.965,E2 -814.965} C_VEL
LIN {X 0,Y 104.638,Z 1200.741,A -85,B 0,C 180,E1 -825.176,E2 -825.176} C_VEL
LIN {X 0,Y 108.868,Z 1199.207,A -85,B 0,C 180,E1 -838.525,E2 -838.525} C_VEL
LIN {X 0,Y 118.537,Z 1195.791,A -85,B 0,C 180,E1 -851.785,E2 -851.785} C_VEL
LIN {X 0,Y 129.964,Z 1191.853,A -85,B 0,C 180,E1 -860.988,E2 -860.988} C_VEL
LIN {X 0,Y 143.958,Z 1186.799,A -85,B 0,C 180,E1 -868.68,E2 -868.68} C_VEL
LIN {X 0,Y 160.728,Z 1180.293,A -85,B 0,C 180,E1 -875.261,E2 -875.261} C_VEL
LIN {X 0,Y 183.315,Z 1170.595,A -85,B 0,C 180,E1 -881.631,E2 -881.631} C_VEL
LIN {X 0,Y 203.179,Z 1160.983,A -85,B 0,C 180,E1 -885.8,E2 -885.8} C_VEL
LIN {X 0,Y 222.083,Z 1150.922,A -85,B 0,C 180,E1 -888.954,E2 -888.954} C_VEL
LIN {X 0,Y 240.61,Z 1140.089,A -85,B 0,C 180,E1 -891.497,E2 -891.497} C_VEL
LIN {X 0,Y 263.376,Z 1125.412,A -85,B 0,C 180,E1 -894.061,E2 -894.061} C_VEL
LIN {X 0,Y 285.61,Z 1109.065,A -85,B 0,C 180,E1 -896.133,E2 -896.133} C_VEL
LIN {X 0,Y 299.305,Z 1098.115,A -85,B 0,C 180,E1 -897.24,E2 -897.24} C_VEL
LIN {X 0,Y 275.986,Z 1116.198,A -85,B 0,C 180,E1 -899.223,E2 -899.223} C_VEL
LIN {X 0,Y 257.014,Z 1129.307,A -85,B 0,C 180,E1 -901.133,E2 -901.133} C_VEL
LIN {X 0,Y 239.343,Z 1140.43,A -85,B 0,C 180,E1 -903.218,E2 -903.218} C_VEL
LIN {X 0,Y 221.089,Z 1150.905,A -85,B 0,C 180,E1 -905.772,E2 -905.772} C_VEL
LIN {X 0,Y 201.392,Z 1161.17,A -85,B 0,C 180,E1 -909.142,E2 -909.142} C_VEL
LIN {X 0,Y 177.576,Z 1172.194,A -85,B 0,C 180,E1 -914.429,E2 -914.429} C_VEL
LIN {X 0,Y 159.44,Z 1179.65,A -85,B 0,C 180,E1 -919.839,E2 -919.839} C_VEL
LIN {X 0,Y 143.689,Z 1185.573,A -85,B 0,C 180,E1 -926.151,E2 -926.151} C_VEL
LIN {X 0,Y 129.326,Z 1190.568,A -85,B 0,C 180,E1 -934.185,E2 -934.185} C_VEL
LIN {X 0,Y 115.6,Z 1195.106,A -85,B 0,C 180,E1 -946.218,E2 -946.218} C_VEL
LIN {X 0,Y 107.585,Z 1197.608,A -85,B 0,C 180,E1 -959.261,E2 -959.261} C_VEL
LIN {X 0,Y 104.603,Z 1198.614,A -85,B 0,C 180,E1 -970.457,E2 -970.457} C_VEL
LIN {X 0,Y 103.943,Z 1198.782,A -85,B 0,C 180,E1 -980.031,E2 -980.031} C_VEL
LIN {X 0,Y 103.938,Z 1198.433,A -85,B 0,C 180,E1 -988.348,E2 -988.348} C_VEL
LIN {X 0,Y 104.628,Z 1197.262,A -85,B 0,C 180,E1 -998.244,E2 -998.244} C_VEL
LIN {X 0,Y 108.646,Z 1194.522,A -85,B 0,C 180,E1 -1011.602,E2 -1011.602} C_VEL
LIN {X 0,Y 116.903,Z 1190.299,A -85,B 0,C 180,E1 -1023.778,E2 -1023.778} C_VEL
LIN {X 0,Y 127.396,Z 1185.433,A -85,B 0,C 180,E1 -1033.067,E2 -1033.067} C_VEL
LIN {X 0,Y 140.413,Z 1179.419,A -85,B 0,C 180,E1 -1040.915,E2 -1040.915} C_VEL
LIN {X 0,Y 157.576,Z 1171.178,A -85,B 0,C 180,E1 -1048.244,E2 -1048.244} C_VEL
LIN {X 0,Y 178.248,Z 1160.28,A -85,B 0,C 180,E1 -1054.574,E2 -1054.574} C_VEL
LIN {X 0,Y 195.468,Z 1150.389,A -85,B 0,C 180,E1 -1058.592,E2 -1058.592} C_VEL
LIN {X 0,Y 212.58,Z 1139.721,A -85,B 0,C 180,E1 -1061.829,E2 -1061.829} C_VEL
LIN {X 0,Y 232.034,Z 1126.487,A -85,B 0,C 180,E1 -1064.855,E2 -1064.855} C_VEL
LIN {X 0,Y 253.851,Z 1109.865,A -85,B 0,C 180,E1 -1067.645,E2 -1067.645} C_VEL
LIN {X 0,Y 271.481,Z 1094.959,A -85,B 0,C 180,E1 -1069.54,E2 -1069.54} C_VEL
LIN {X 0,Y 287.476,Z 1080.156,A -85,B 0,C 180,E1 -1071.04,E2 -1071.04} C_VEL
LIN {X 0,Y 304.598,Z 1062.773,A -85,B 0,C 180,E1 -1072.462,E2 -1072.462} C_VEL
LIN {X 0,Y 323.329,Z 1041.398,A -85,B 0,C 180,E1 -1073.842,E2 -1073.842} C_VEL
LIN {X 0,Y 337.362,Z 1023.501,A -85,B 0,C 180,E1 -1074.776,E2 -1074.776} C_VEL
LIN {X 0,Y 350.508,Z 1004.971,A -85,B 0,C 180,E1 -1075.568,E2 -1075.568} C_VEL
LIN {X 0,Y 362.73,Z 985.837,A -85,B 0,C 180,E1 -1076.262,E2 -1076.262} C_VEL
LIN {X 0,Y 375.17,Z 964.024,A -85,B 0,C 180,E1 -1076.913,E2 -1076.913} C_VEL
LIN {X 0,Y 369.423,Z 974.4,A -85,B 0,C 180,E1 -1077.193,E2 -1077.193} C_VEL
LIN {X 0,Y 364.199,Z 983.593,A -85,B 0,C 180,E1 -1077.304,E2 -1077.304} C_VEL
LIN {X 0,Y 350.041,Z 1005.971,A -85,B 0,C 180,E1 -1077.087,E2 -1077.087} C_VEL
LIN {X 0,Y 343.937,Z 1014.536,A -85,B 0,C 180,E1 -1077.227,E2 -1077.227} C_VEL
LIN {X 0,Y 343.494,Z 1015.129,A -85,B 0,C 180,E1 -1077.25,E2 -1077.25} C_VEL
LIN {X 0,Y 327.424,Z 1036.155,A -85,B 0,C 180,E1 -1078.163,E2 -1078.163} C_VEL
LIN {X 0,Y 312.908,Z 1053.316,A -85,B 0,C 180,E1 -1079.084,E2 -1079.084} C_VEL
LIN {X 0,Y 297.967,Z 1069.404,A -85,B 0,C 180,E1 -1080.139,E2 -1080.139} C_VEL
LIN {X 0,Y 279.577,Z 1087.413,A -85,B 0,C 180,E1 -1081.599,E2 -1081.599} C_VEL
LIN {X 0,Y 258.446,Z 1105.76,A -85,B 0,C 180,E1 -1083.549,E2 -1083.549} C_VEL
LIN {X 0,Y 241.055,Z 1119.412,A -85,B 0,C 180,E1 -1085.431,E2 -1085.431} C_VEL
LIN {X 0,Y 223.942,Z 1131.707,A -85,B 0,C 180,E1 -1087.599,E2 -1087.599} C_VEL
LIN {X 0,Y 204.449,Z 1144.51,A -85,B 0,C 180,E1 -1090.572,E2 -1090.572} C_VEL
LIN {X 0,Y 181.217,Z 1158.16,A -85,B 0,C 180,E1 -1095.074,E2 -1095.074} C_VEL
LIN {X 0,Y 163.414,Z 1167.603,A -85,B 0,C 180,E1 -1099.56,E2 -1099.56} C_VEL
LIN {X 0,Y 146.771,Z 1175.765,A -85,B 0,C 180,E1 -1105.03,E2 -1105.03} C_VEL
LIN {X 0,Y 130.33,Z 1183.333,A -85,B 0,C 180,E1 -1112.442,E2 -1112.442} C_VEL
LIN {X 0,Y 113.465,Z 1190.72,A -85,B 0,C 180,E1 -1124.121,E2 -1124.121} C_VEL
LIN {X 0,Y 104.18,Z 1194.917,A -85,B 0,C 180,E1 -1134.838,E2 -1134.838} C_VEL
LIN {X 0,Y 98.667,Z 1197.828,A -85,B 0,C 180,E1 -1146.084,E2 -1146.084} C_VEL
LIN {X 0,Y 96.275,Z 1199.723,A -85,B 0,C 180,E1 -1157.493,E2 -1157.493} C_VEL
LIN {X 0,Y 95.914,Z 1200.674,A -85,B 0,C 180,E1 -1167.01,E2 -1167.01} C_VEL
LIN {X 0,Y 95.921,Z 1200.96,A -85,B 0,C 180,E1 -1174.781,E2 -1174.781} C_VEL
LIN {X 0,Y 96.583,Z 1200.721,A -85,B 0,C 180,E1 -1184.997,E2 -1184.997} C_VEL
LIN {X 0,Y 99.945,Z 1199.606,A -85,B 0,C 180,E1 -1197.077,E2 -1197.077} C_VEL
LIN {X 0,Y 108.73,Z 1196.975,A -85,B 0,C 180,E1 -1210.759,E2 -1210.759} C_VEL
LIN {X 0,Y 123.783,Z 1192.21,A -85,B 0,C 180,E1 -1223.291,E2 -1223.291} C_VEL
LIN {X 0,Y 139.058,Z 1187.067,A -85,B 0,C 180,E1 -1231.305,E2 -1231.305} C_VEL
LIN {X 0,Y 155.802,Z 1180.932,A -85,B 0,C 180,E1 -1237.535,E2 -1237.535} C_VEL
LIN {X 0,Y 176.791,Z 1172.447,A -85,B 0,C 180,E1 -1243.235,E2 -1243.235} C_VEL
LIN {X 0,Y 200.383,Z 1161.541,A -85,B 0,C 180,E1 -1247.955,E2 -1247.955} C_VEL
LIN {X 0,Y 219.701,Z 1151.56,A -85,B 0,C 180,E1 -1250.954,E2 -1250.954} C_VEL
LIN {X 0,Y 238.567,Z 1140.808,A -85,B 0,C 180,E1 -1253.359,E2 -1253.359} C_VEL
LIN {X 0,Y 257.793,Z 1128.74,A -85,B 0,C 180,E1 -1255.402,E2 -1255.402} C_VEL
LIN {X 0,Y 278.5,Z 1114.395,A -85,B 0,C 180,E1 -1257.255,E2 -1257.255} C_VEL
LIN {X 0,Y 256.988,Z 1129.115,A -85,B 0,C 180,E1 -1259.212,E2 -1259.212} C_VEL
LIN {X 0,Y 238.024,Z 1140.848,A -85,B 0,C 180,E1 -1261.262,E2 -1261.262} C_VEL
LIN {X 0,Y 219.416,Z 1151.289,A -85,B 0,C 180,E1 -1263.663,E2 -1263.663} C_VEL
LIN {X 0,Y 197.512,Z 1162.388,A -85,B 0,C 180,E1 -1267.163,E2 -1267.163} C_VEL
LIN {X 0,Y 173.839,Z 1172.838,A -85,B 0,C 180,E1 -1272.104,E2 -1272.104} C_VEL
LIN {X 0,Y 155.613,Z 1180.007,A -85,B 0,C 180,E1 -1277.192,E2 -1277.192} C_VEL
LIN {X 0,Y 138.587,Z 1186.061,A -85,B 0,C 180,E1 -1283.616,E2 -1283.616} C_VEL
LIN {X 0,Y 120.919,Z 1191.809,A -85,B 0,C 180,E1 -1293.371,E2 -1293.371} C_VEL
LIN {X 0,Y 107.138,Z 1195.764,A -85,B 0,C 180,E1 -1305.941,E2 -1305.941} C_VEL
LIN {X 0,Y 99.917,Z 1197.801,A -85,B 0,C 180,E1 -1317.972,E2 -1317.972} C_VEL
LIN {X 0,Y 96.727,Z 1198.715,A -85,B 0,C 180,E1 -1329.426,E2 -1329.426} C_VEL
LIN {X 0,Y 95.946,Z 1198.857,A -85,B 0,C 180,E1 -1339.798,E2 -1339.798} C_VEL
LIN {X 0,Y 95.936,Z 1198.531,A -85,B 0,C 180,E1 -1348.211,E2 -1348.211} C_VEL
LIN {X 0,Y 96.702,Z 1197.38,A -85,B 0,C 180,E1 -1358.925,E2 -1358.925} C_VEL
LIN {X 0,Y 101.195,Z 1194.681,A -85,B 0,C 180,E1 -1373.282,E2 -1373.282} C_VEL
LIN {X 0,Y 110.446,Z 1190.394,A -85,B 0,C 180,E1 -1386.318,E2 -1386.318} C_VEL
LIN {X 0,Y 121.58,Z 1185.633,A -85,B 0,C 180,E1 -1395.686,E2 -1395.686} C_VEL
LIN {X 0,Y 134.746,Z 1179.938,A -85,B 0,C 180,E1 -1403.267,E2 -1403.267} C_VEL
LIN {X 0,Y 150.414,Z 1172.805,A -85,B 0,C 180,E1 -1409.791,E2 -1409.791} C_VEL
LIN {X 0,Y 170.805,Z 1162.816,A -85,B 0,C 180,E1 -1415.955,E2 -1415.955} C_VEL
LIN {X 0,Y 191.777,Z 1151.208,A -85,B 0,C 180,E1 -1420.683,E2 -1420.683} C_VEL
LIN {X 0,Y 209.29,Z 1140.623,A -85,B 0,C 180,E1 -1423.798,E2 -1423.798} C_VEL
LIN {X 0,Y 226.394,Z 1129.34,A -85,B 0,C 180,E1 -1426.324,E2 -1426.324} C_VEL
LIN {X 0,Y 245.953,Z 1115.201,A -85,B 0,C 180,E1 -1428.747,E2 -1428.747} C_VEL
LIN {X 0,Y 267.293,Z 1097.891,A -85,B 0,C 180,E1 -1430.961,E2 -1430.961} C_VEL
LIN {X 0,Y 284.415,Z 1082.454,A -85,B 0,C 180,E1 -1432.479,E2 -1432.479} C_VEL
LIN {X 0,Y 299.782,Z 1067.271,A -85,B 0,C 180,E1 -1433.69,E2 -1433.69} C_VEL
LIN {X 0,Y 315.267,Z 1050.486,A -85,B 0,C 180,E1 -1434.79,E2 -1434.79} C_VEL
LIN {X 0,Y 333.303,Z 1028.739,A -85,B 0,C 180,E1 -1435.928,E2 -1435.928} C_VEL
LIN {X 0,Y 348.506,Z 1007.84,A -85,B 0,C 180,E1 -1436.792,E2 -1436.792} C_VEL
LIN {X 0,Y 350.099,Z 1005.502,A -85,B 0,C 180,E1 -1436.889,E2 -1436.889} C_VEL
LIN {X 0,Y 343.494,Z 1015.129,A -85,B 0,C 180,E1 -1437.25,E2 -1437.25} C_VEL
LIN {X 0,Y 338.025,Z 1022.456,A -85,B 0,C 180,E1 -1437.382,E2 -1437.382} C_VEL
LIN {X 0,Y 323.43,Z 1041.044,A -85,B 0,C 180,E1 -1437.144,E2 -1437.144} C_VEL
LIN {X 0,Y 317.489,Z 1047.911,A -85,B 0,C 180,E1 -1437.305,E2 -1437.305} C_VEL
LIN {X 0,Y 301.094,Z 1065.77,A -85,B 0,C 180,E1 -1438.325,E2 -1438.325} C_VEL
LIN {X 0,Y 284.981,Z 1081.714,A -85,B 0,C 180,E1 -1439.45,E2 -1439.45} C_VEL
LIN {X 0,Y 267.996,Z 1097.021,A -85,B 0,C 180,E1 -1440.801,E2 -1440.801} C_VEL
LIN {X 0,Y 246.587,Z 1114.485,A -85,B 0,C 180,E1 -1442.789,E2 -1442.789} C_VEL
LIN {X 0,Y 225.866,Z 1129.39,A -85,B 0,C 180,E1 -1445.09,E2 -1445.09} C_VEL
LIN {X 0,Y 207.764,Z 1141.236,A -85,B 0,C 180,E1 -1447.518,E2 -1447.518} C_VEL
LIN {X 0,Y 190.091,Z 1151.799,A -85,B 0,C 180,E1 -1450.38,E2 -1450.38} C_VEL
LIN {X 0,Y 170.317,Z 1162.579,A -85,B 0,C 180,E1 -1454.378,E2 -1454.378} C_VEL
LIN {X 0,Y 147.296,Z 1173.776,A -85,B 0,C 180,E1 -1460.671,E2 -1460.671} C_VEL
LIN {X 0,Y 130.352,Z 1181.248,A -85,B 0,C 180,E1 -1467.15,E2 -1467.15} C_VEL
LIN {X 0,Y 115.895,Z 1187.25,A -85,B 0,C 180,E1 -1474.952,E2 -1474.952} C_VEL
LIN {X 0,Y 103.35,Z 1192.34,A -85,B 0,C 180,E1 -1485.066,E2 -1485.066} C_VEL
LIN {X 0,Y 93.032,Z 1196.873,A -85,B 0,C 180,E1 -1499.657,E2 -1499.657} C_VEL
LIN {X 0,Y 88.543,Z 1199.457,A -85,B 0,C 180,E1 -1514.943,E2 -1514.943} C_VEL
LIN {X 0,Y 87.919,Z 1200.532,A -85,B 0,C 180,E1 -1525.431,E2 -1525.431} C_VEL
LIN {X 0,Y 87.912,Z 1200.8,A -85,B 0,C 180,E1 -1533.257,E2 -1533.257} C_VEL
LIN {X 0,Y 88.265,Z 1200.79,A -85,B 0,C 180,E1 -1542.427,E2 -1542.427} C_VEL
LIN {X 0,Y 91.065,Z 1200.001,A -85,B 0,C 180,E1 -1555.351,E2 -1555.351} C_VEL
LIN {X 0,Y 98.083,Z 1198.087,A -85,B 0,C 180,E1 -1568.448,E2 -1568.448} C_VEL
LIN {X 0,Y 108.939,Z 1195.096,A -85,B 0,C 180,E1 -1579.62,E2 -1579.62} C_VEL
LIN {X 0,Y 122.866,Z 1191.012,A -85,B 0,C 180,E1 -1588.699,E2 -1588.699} C_VEL
LIN {X 0,Y 141.447,Z 1185.047,A -85,B 0,C 180,E1 -1596.77,E2 -1596.77} C_VEL
LIN {X 0,Y 164.658,Z 1176.475,A -85,B 0,C 180,E1 -1603.621,E2 -1603.621} C_VEL
LIN {X 0,Y 184.141,Z 1168.342,A -85,B 0,C 180,E1 -1607.786,E2 -1607.786} C_VEL
LIN {X 0,Y 202.772,Z 1159.708,A -85,B 0,C 180,E1 -1610.921,E2 -1610.921} C_VEL
LIN {X 0,Y 222.358,Z 1149.648,A -85,B 0,C 180,E1 -1613.59,E2 -1613.59} C_VEL
LIN {X 0,Y 245.523,Z 1136.42,A -85,B 0,C 180,E1 -1616.135,E2 -1616.135} C_VEL
LIN {X 0,Y 257.471,Z 1128.783,A -85,B 0,C 180,E1 -1617.27,E2 -1617.27} C_VEL
LIN {X 0,Y 237.99,Z 1140.683,A -85,B 0,C 180,E1 -1619.178,E2 -1619.178} C_VEL
LIN {X 0,Y 219.033,Z 1151.15,A -85,B 0,C 180,E1 -1621.398,E2 -1621.398} C_VEL
LIN {X 0,Y 197.577,Z 1161.809,A -85,B 0,C 180,E1 -1624.488,E2 -1624.488} C_VEL
LIN {X 0,Y 172.226,Z 1172.772,A -85,B 0,C 180,E1 -1629.275,E2 -1629.275} C_VEL
LIN {X 0,Y 153.542,Z 1179.863,A -85,B 0,C 180,E1 -1634.006,E2 -1634.006} C_VEL
LIN {X 0,Y 136.133,Z 1185.781,A -85,B 0,C 180,E1 -1639.93,E2 -1639.93} C_VEL
LIN {X 0,Y 119.776,Z 1190.772,A -85,B 0,C 180,E1 -1647.768,E2 -1647.768} C_VEL
LIN {X 0,Y 103.04,Z 1195.38,A -85,B 0,C 180,E1 -1660.554,E2 -1660.554} C_VEL
LIN {X 0,Y 93.106,Z 1197.809,A -85,B 0,C 180,E1 -1674.705,E2 -1674.705} C_VEL
LIN {X 0,Y 88.997,Z 1198.796,A -85,B 0,C 180,E1 -1687.546,E2 -1687.546} C_VEL
LIN {X 0,Y 87.959,Z 1198.956,A -85,B 0,C 180,E1 -1698.86,E2 -1698.86} C_VEL
LIN {X 0,Y 87.923,Z 1198.651,A -85,B 0,C 180,E1 -1707.395,E2 -1707.395} C_VEL
LIN {X 0,Y 88.517,Z 1197.697,A -85,B 0,C 180,E1 -1717.793,E2 -1717.793} C_VEL
LIN {X 0,Y 91.672,Z 1195.776,A -85,B 0,C 180,E1 -1730.43,E2 -1730.43} C_VEL
LIN {X 0,Y 100.121,Z 1192.186,A -85,B 0,C 180,E1 -1744.7,E2 -1744.7} C_VEL
LIN {X 0,Y 114.818,Z 1186.33,A -85,B 0,C 180,E1 -1757.752,E2 -1757.752} C_VEL
LIN {X 0,Y 129.325,Z 1180.456,A -85,B 0,C 180,E1 -1765.822,E2 -1765.822} C_VEL
LIN {X 0,Y 144.919,Z 1173.74,A -85,B 0,C 180,E1 -1772.027,E2 -1772.027} C_VEL
LIN {X 0,Y 162.619,Z 1165.484,A -85,B 0,C 180,E1 -1777.266,E2 -1777.266} C_VEL
LIN {X 0,Y 185.715,Z 1153.54,A -85,B 0,C 180,E1 -1782.359,E2 -1782.359} C_VEL
LIN {X 0,Y 206.256,Z 1141.521,A -85,B 0,C 180,E1 -1785.828,E2 -1785.828} C_VEL
LIN {X 0,Y 224.607,Z 1129.7,A -85,B 0,C 180,E1 -1788.344,E2 -1788.344} C_VEL
LIN {X 0,Y 243.316,Z 1116.448,A -85,B 0,C 180,E1 -1790.492,E2 -1790.492} C_VEL
LIN {X 0,Y 266.137,Z 1098.341,A -85,B 0,C 180,E1 -1792.684,E2 -1792.684} C_VEL
LIN {X 0,Y 283.993,Z 1082.443,A -85,B 0,C 180,E1 -1794.14,E2 -1794.14} C_VEL
LIN {X 0,Y 299.491,Z 1067.289,A -85,B 0,C 180,E1 -1795.258,E2 -1795.258} C_VEL
LIN {X 0,Y 315.026,Z 1050.61,A -85,B 0,C 180,E1 -1796.272,E2 -1796.272} C_VEL
LIN {X 0,Y 324.952,Z 1039.013,A -85,B 0,C 180,E1 -1796.867,E2 -1796.867} C_VEL
LIN {X 0,Y 317.489,Z 1047.911,A -85,B 0,C 180,E1 -1797.305,E2 -1797.305} C_VEL
LIN {X 0,Y 311.969,Z 1054.059,A -85,B 0,C 180,E1 -1797.448,E2 -1797.448} C_VEL
LIN {X 0,Y 297.307,Z 1069.681,A -85,B 0,C 180,E1 -1797.195,E2 -1797.195} C_VEL
LIN {X 0,Y 291.406,Z 1075.423,A -85,B 0,C 180,E1 -1797.364,E2 -1797.364} C_VEL
LIN {X 0,Y 271.634,Z 1093.456,A -85,B 0,C 180,E1 -1798.734,E2 -1798.734} C_VEL
LIN {X 0,Y 254.972,Z 1107.264,A -85,B 0,C 180,E1 -1800.065,E2 -1800.065} C_VEL
LIN {X 0,Y 237.079,Z 1120.777,A -85,B 0,C 180,E1 -1801.71,E2 -1801.71} C_VEL
LIN {X 0,Y 216.48,Z 1134.889,A -85,B 0,C 180,E1 -1803.973,E2 -1803.973} C_VEL
LIN {X 0,Y 193.368,Z 1148.903,A -85,B 0,C 180,E1 -1807.129,E2 -1807.129} C_VEL
LIN {X 0,Y 173.89,Z 1159.47,A -85,B 0,C 180,E1 -1810.493,E2 -1810.493} C_VEL
LIN {X 0,Y 155.632,Z 1168.458,A -85,B 0,C 180,E1 -1814.511,E2 -1814.511} C_VEL
LIN {X 0,Y 136.243,Z 1177.136,A -85,B 0,C 180,E1 -1820.178,E2 -1820.178} C_VEL
LIN {X 0,Y 114.794,Z 1185.747,A -85,B 0,C 180,E1 -1829.419,E2 -1829.419} C_VEL
LIN {X 0,Y 100.472,Z 1191.102,A -85,B 0,C 180,E1 -1839.079,E2 -1839.079} C_VEL
LIN {X 0,Y 89.811,Z 1195.098,A -85,B 0,C 180,E1 -1850.608,E2 -1850.608} C_VEL
LIN {X 0,Y 83.154,Z 1197.908,A -85,B 0,C 180,E1 -1863.58,E2 -1863.58} C_VEL
LIN {X 0,Y 80.358,Z 1199.621,A -85,B 0,C 180,E1 -1876.322,E2 -1876.322} C_VEL
LIN {X 0,Y 79.913,Z 1200.504,A -85,B 0,C 180,E1 -1887.128,E2 -1887.128} C_VEL
LIN {X 0,Y 79.934,Z 1200.767,A -85,B 0,C 180,E1 -1895.74,E2 -1895.74} C_VEL
LIN {X 0,Y 81.003,Z 1200.557,A -85,B 0,C 180,E1 -1908.105,E2 -1908.105} C_VEL
LIN {X 0,Y 85.457,Z 1199.517,A -85,B 0,C 180,E1 -1921.767,E2 -1921.767} C_VEL
LIN {X 0,Y 95.166,Z 1197.234,A -85,B 0,C 180,E1 -1935.595,E2 -1935.595} C_VEL
LIN {X 0,Y 113.689,Z 1192.457,A -85,B 0,C 180,E1 -1949.525,E2 -1949.525} C_VEL
LIN {X 0,Y 131.844,Z 1187.09,A -85,B 0,C 180,E1 -1957.716,E2 -1957.716} C_VEL
LIN {X 0,Y 150.19,Z 1181.003,A -85,B 0,C 180,E1 -1963.464,E2 -1963.464} C_VEL
LIN {X 0,Y 170.6,Z 1173.374,A -85,B 0,C 180,E1 -1968.167,E2 -1968.167} C_VEL
LIN {X 0,Y 197.571,Z 1161.749,A -85,B 0,C 180,E1 -1972.705,E2 -1972.705} C_VEL
LIN {X 0,Y 218.67,Z 1151.305,A -85,B 0,C 180,E1 -1975.409,E2 -1975.409} C_VEL
LIN {X 0,Y 236.229,Z 1141.683,A -85,B 0,C 180,E1 -1977.298,E2 -1977.298} C_VEL
LIN {X 0,Y 214.974,Z 1153.101,A -85,B 0,C 180,E1 -1979.606,E2 -1979.606} C_VEL
LIN {X 0,Y 189.26,Z 1165.183,A -85,B 0,C 180,E1 -1983.163,E2 -1983.163} C_VEL
LIN {X 0,Y 168.218,Z 1173.778,A -85,B 0,C 180,E1 -1986.969,E2 -1986.969} C_VEL
LIN {X 0,Y 148.987,Z 1180.737,A -85,B 0,C 180,E1 -1991.536,E2 -1991.536} C_VEL
LIN {X 0,Y 129.105,Z 1187.095,A -85,B 0,C 180,E1 -1998.047,E2 -1998.047} C_VEL
LIN {X 0,Y 107.472,Z 1192.999,A -85,B 0,C 180,E1 -2009.014,E2 -2009.014} C_VEL
LIN {X 0,Y 94.066,Z 1196.172,A -85,B 0,C 180,E1 -2020.422,E2 -2020.422} C_VEL
LIN {X 0,Y 85.395,Z 1198.056,A -85,B 0,C 180,E1 -2033.337,E2 -2033.337} C_VEL
LIN {X 0,Y 81.081,Z 1198.918,A -85,B 0,C 180,E1 -2046.761,E2 -2046.761} C_VEL
LIN {X 0,Y 79.967,Z 1199.031,A -85,B 0,C 180,E1 -2058.463,E2 -2058.463} C_VEL
LIN {X 0,Y 79.929,Z 1198.726,A -85,B 0,C 180,E1 -2067.852,E2 -2067.852} C_VEL
LIN {X 0,Y 80.683,Z 1197.747,A -85,B 0,C 180,E1 -2079.274,E2 -2079.274} C_VEL
LIN {X 0,Y 84.735,Z 1195.692,A -85,B 0,C 180,E1 -2093.656,E2 -2093.656} C_VEL
LIN {X 0,Y 96.056,Z 1191.442,A -85,B 0,C 180,E1 -2110.197,E2 -2110.197} C_VEL
LIN {X 0,Y 110.825,Z 1186.034,A -85,B 0,C 180,E1 -2121.717,E2 -2121.717} C_VEL
LIN {X 0,Y 126.419,Z 1180.085,A -85,B 0,C 180,E1 -2129.557,E2 -2129.557} C_VEL
LIN {X 0,Y 143.715,Z 1172.947,A -85,B 0,C 180,E1 -2135.705,E2 -2135.705} C_VEL
LIN {X 0,Y 165.744,Z 1162.923,A -85,B 0,C 180,E1 -2141.353,E2 -2141.353} C_VEL
LIN {X 0,Y 187.919,Z 1151.329,A -85,B 0,C 180,E1 -2145.558,E2 -2145.558} C_VEL
LIN {X 0,Y 206.266,Z 1140.731,A -85,B 0,C 180,E1 -2148.297,E2 -2148.297} C_VEL
LIN {X 0,Y 224.991,Z 1128.814,A -85,B 0,C 180,E1 -2150.61,E2 -2150.61} C_VEL
LIN {X 0,Y 246.896,Z 1113.38,A -85,B 0,C 180,E1 -2152.843,E2 -2152.843} C_VEL
LIN {X 0,Y 268.136,Z 1096.3,A -85,B 0,C 180,E1 -2154.654,E2 -2154.654} C_VEL
LIN {X 0,Y 284.708,Z 1081.597,A -85,B 0,C 180,E1 -2155.867,E2 -2155.867} C_VEL
LIN {X 0,Y 299.628,Z 1067.102,A -85,B 0,C 180,E1 -2156.846,E2 -2156.846} C_VEL
LIN {X 0,Y 291.406,Z 1075.423,A -85,B 0,C 180,E1 -2157.364,E2 -2157.364} C_VEL
LIN {X 0,Y 285.728,Z 1080.761,A -85,B 0,C 180,E1 -2157.525,E2 -2157.525} C_VEL
LIN {X 0,Y 270.707,Z 1094.097,A -85,B 0,C 180,E1 -2157.262,E2 -2157.262} C_VEL
LIN {X 0,Y 264.864,Z 1099.026,A -85,B 0,C 180,E1 -2157.452,E2 -2157.452} C_VEL
LIN {X 0,Y 241.362,Z 1117.25,A -85,B 0,C 180,E1 -2159.288,E2 -2159.288} C_VEL
LIN {X 0,Y 222.784,Z 1130.109,A -85,B 0,C 180,E1 -2161.029,E2 -2161.029} C_VEL
LIN {X 0,Y 204.276,Z 1141.733,A -85,B 0,C 180,E1 -2163.095,E2 -2163.095} C_VEL
LIN {X 0,Y 184.903,Z 1152.754,A -85,B 0,C 180,E1 -2165.725,E2 -2165.725} C_VEL
LIN {X 0,Y 160.201,Z 1165.253,A -85,B 0,C 180,E1 -2170.065,E2 -2170.065} C_VEL
LIN {X 0,Y 139.729,Z 1174.321,A -85,B 0,C 180,E1 -2174.97,E2 -2174.97} C_VEL
LIN {X 0,Y 121.942,Z 1181.433,A -85,B 0,C 180,E1 -2180.807,E2 -2180.807} C_VEL
LIN {X 0,Y 105.705,Z 1187.378,A -85,B 0,C 180,E1 -2188.39,E2 -2188.39} C_VEL
LIN {X 0,Y 88.789,Z 1193.26,A -85,B 0,C 180,E1 -2201.014,E2 -2201.014} C_VEL
